# B&R Automation Studio project PLC code - cp (part 4)

#### ResetComms.st
```iecst
ACTION ResetComms:

	CanGetState.enable := TRUE;
	CanGetState.node := dataInv.Parameters.Hardware.Node;
	CanGetState.pDevice := ADR('SS1.IF1');
	CanGetState();

	iReasonNotComms.0 := CanGetState.state = coPREOPERATIONAL;
	iReasonNotComms.1 := CanGetState.state = coUNKNOWN;
	iReasonNotComms.2 := CanGetState.state = coNOTAVAIL;
	iReasonNotComms.3 := dataInv.Status.ErrorComms;

	tonNotComms.IN := iReasonNotComms > 0;
	tonNotComms.PT := t#3s;
	tonNotComms();

	xChangedResetCommsState := CanResetState_copy <> CanResetState;
	CanResetState_copy := CanResetState;

	CASE CanResetState OF

		COCOMSR_UNDEFINED,
		COCOMSR_COMMUNICATING:

			iTimesTryToReset := 0;

			//If time in error, define an error comms
			IF tonNotComms.Q THEN
				CanResetState := COCOMSR_COMMSERROR;
			END_IF

		COCOMSR_COMMSERROR:
			//Start the resetting process
			IF dataInv.Commands.Reset THEN //AND dataInv.Parameter.xAutoresetComms THEN
				//Communication has returned to work
				IF CanGetState.state = coOPERATIONAL THEN
					CanResetState := COCOMSR_COMMUNICATING;
				ELSE
					CanResetState := COCOMSR_RESETTING;
				END_IF
			END_IF

		COCOMSR_RESETTING:
			CANopenReset.enable := TRUE;
			CANopenReset.node := dataInv.Parameters.Hardware.Node;
			CANopenReset.pDevice := ADR('SS1.IF1');
			CANopenReset.state := coRESET_NODE;
			CANopenReset();

			IF CANopenReset.status = ERR_OK THEN
				lastCanOpenResetError := CANopenReset.error;
				CANopenReset(enable := FALSE);
				CanResetState := COCOMSR_WAITINGTOBERESETTED;
			END_IF

			tonCommsErrorResetting.IN := NOT xChangedResetCommsState;
			tonCommsErrorResetting.PT := t#10s;
			tonCommsErrorResetting();

			IF tonCommsErrorResetting.Q THEN
				lastResetingState := CanGetState.state;
				lastFbResetStatus := CANopenReset.status;
				tonCommsErrorResetting(IN:=FALSE);
				CANopenReset(enable:=FALSE);
				CanResetState := COCOMSR_RESETTING_ERROR;
			END_IF

		COCOMSR_WAITINGTOBERESETTED:

			//Communication has returned to work
			IF CanGetState.state = coOPERATIONAL THEN
				CanResetState := COCOMSR_COMMUNICATING;
			END_IF

			tonCommsErrorResetting.IN := NOT xChangedResetCommsState;
			tonCommsErrorResetting.PT := t#4s;
			tonCommsErrorResetting();

			IF tonCommsErrorResetting.Q THEN
				lastResetingState := CanGetState.state;
				lastFbResetStatus := CANopenReset.status;
				tonCommsErrorResetting(IN:=FALSE);
				CanResetState := COCOMSR_RESETTING_ERROR;
			END_IF

		COCOMSR_RESETTING_ERROR:

			//After an error, wait to try again
			tonCommsErrorResetting.IN := NOT xChangedResetCommsState;
			tonCommsErrorResetting.PT := t#500ms;
			tonCommsErrorResetting();

			IF tonCommsErrorResetting.Q  AND iTimesTryToReset < 6 THEN
				iTimesTryToReset := iTimesTryToReset + 1;
				CanResetState := COCOMSR_RESETTING;
			ELSIF tonCommsErrorResetting.Q THEN
				CanResetState := COCOMSR_COMMSERROR;
			END_IF

	END_CASE;

END_ACTION
```

#### Simulation.st
```iecst
ACTION Simulation:

	dataInv.Status.ErrorComms := FALSE;
	(********** Reset non appliant in simulation error flags **********)
	paramOk := TRUE;
	invalidHwAddress := FALSE;
	ioMap.In.ModuleOk := TRUE;
	connectionErrorNotAck := FALSE; //Uncomment for P66/P76
	(********** Inverter state machine **********)
	CASE StepSim OF
		STATE_NOT_READY_TO_SWITCH_ON:
			ioMap.In.StatusWord := 16#0000;
			IF ioMap.Out.ControlWord = 16#0000 THEN
				StepSim := STATE_SWITCH_ON_DISABLED;
			END_IF;

		STATE_SWITCH_ON_DISABLED:
			ioMap.In.StatusWord := 16#0040;
			IF ioMap.Out.ControlWord = 16#0006 THEN
				StepSim := STATE_READY_TO_SWITCH_ON;
			END_IF;

		STATE_READY_TO_SWITCH_ON:
			ioMap.In.StatusWord := 16#0021;
			IF ioMap.Out.ControlWord = 16#0007 THEN
				StepSim := STATE_SWITCHED_ON;
			ELSIF ioMap.Out.ControlWord = 16#0000 OR ioMap.Out.ControlWord = 16#0002 THEN
				StepSim := STATE_SWITCH_ON_DISABLED;
			END_IF;

		STATE_SWITCHED_ON:
			ioMap.In.StatusWord := 16#0023;
			IF ioMap.Out.ControlWord = 16#000F THEN
				StepSim := STATE_OPERATION_ENABLED;
			ELSIF ioMap.Out.ControlWord = 16#0006 THEN
				StepSim := STATE_READY_TO_SWITCH_ON;
			ELSIF ioMap.Out.ControlWord = 16#0000 OR ioMap.Out.ControlWord = 16#0002 THEN
				StepSim := STATE_SWITCH_ON_DISABLED;
			END_IF;

		STATE_OPERATION_ENABLED:
			ioMap.In.StatusWord := 16#0027;
			IF ioMap.Out.ControlWord = 16#0007 THEN
				StepSim := STATE_SWITCHED_ON;
			ELSIF ioMap.Out.ControlWord = 16#0006 THEN
				StepSim := STATE_READY_TO_SWITCH_ON;
			ELSIF ioMap.Out.ControlWord = 16#0000 OR ioMap.Out.ControlWord = 16#0002 THEN
				StepSim := STATE_SWITCH_ON_DISABLED;
			END_IF;

		STATE_QUICK_STOP_ACTIVE:
			ioMap.In.StatusWord := 16#0007;
			IF ioMap.Out.ControlWord = 16#0000 OR ioMap.Out.ControlWord = 16#0002 THEN
				StepSim := STATE_SWITCH_ON_DISABLED;
			END_IF;

		STATE_FAULT_REACTION_ACTIVE:
			ioMap.In.StatusWord := 16#000F;
			StepSim := STATE_FAULT;

		STATE_FAULT:
			ioMap.In.StatusWord := 16#0008;
			IF ioMap.Out.ControlWord = 16#0080 THEN
				StepSim := STATE_SWITCH_ON_DISABLED;
			END_IF;
	END_CASE;
	(********** Movement profile **********)
	IF StepSim = STATE_OPERATION_ENABLED THEN
		(* No decceleration parameter involved during operation *)
		SimDecceleration := 0;
		(* Acceleration and velocity calculation *)
		IF direction = 1 THEN
			IF REAL_TO_INT(SimVelocity) = UINT_TO_INT(dataInv.Parameters.Velocity) THEN
				SimAcceleration := 0;
			ELSIF REAL_TO_INT(SimVelocity) < UINT_TO_INT(dataInv.Parameters.Velocity) THEN
				SimAcceleration := UINT_TO_REAL(SimNominalSpeed) / dataInv.Parameters.AccelerationTime; (* positive acceleration in positive direction *)
				SimVelocity := LIMIT(-1*UINT_TO_REAL(SimNominalSpeed), SimInitialVelocity + SimVelocity + direction*(SimAcceleration * SimCycleTime), UINT_TO_REAL(dataInv.Parameters.Velocity));
			ELSIF REAL_TO_INT(SimVelocity) > UINT_TO_INT(dataInv.Parameters.Velocity) THEN
				SimAcceleration := -1*(UINT_TO_REAL(SimNominalSpeed) / dataInv.Parameters.AccelerationTime); (* negative acceleration in positive direction *)
				SimVelocity := LIMIT(UINT_TO_REAL(dataInv.Parameters.Velocity), SimInitialVelocity + SimVelocity + direction*(SimAcceleration * SimCycleTime), UINT_TO_REAL(SimNominalSpeed));
			END_IF;
		ELSIF direction = -1 THEN
			IF REAL_TO_INT(SimVelocity) = direction*UINT_TO_INT(dataInv.Parameters.Velocity) THEN
				SimAcceleration := 0;
			ELSIF REAL_TO_INT(SimVelocity) > direction*UINT_TO_INT(dataInv.Parameters.Velocity) THEN
				SimAcceleration := UINT_TO_REAL(SimNominalSpeed) / dataInv.Parameters.AccelerationTime; (* positive acceleration in negative direction *)
				SimVelocity := LIMIT(-1*UINT_TO_REAL(dataInv.Parameters.Velocity), SimInitialVelocity + SimVelocity + direction*(SimAcceleration * SimCycleTime), UINT_TO_REAL(SimNominalSpeed));
			ELSIF REAL_TO_INT(SimVelocity) < direction*UINT_TO_INT(dataInv.Parameters.Velocity) THEN
				SimAcceleration := -1*(UINT_TO_REAL(SimNominalSpeed) / dataInv.Parameters.AccelerationTime); (* negative acceleration in negative direction *)
				SimVelocity := LIMIT(-1*UINT_TO_REAL(SimNominalSpeed), SimInitialVelocity + SimVelocity + direction*(SimAcceleration * SimCycleTime), -1*UINT_TO_REAL(dataInv.Parameters.Velocity));
			END_IF;
		END_IF;
		(* Limiting the velocity to the nominal speed of the motor - Optional *)
		SimVelocity := LIMIT(-1*UINT_TO_REAL(SimNominalSpeed),SimVelocity,UINT_TO_REAL(SimNominalSpeed));

	ELSE
		(* No acceleration parameter involved during stop *)
		SimAcceleration := 0;
		(* Decceleration and velocity calculation *)
		IF REAL_TO_INT(SimVelocity) = 0 THEN
			SimDecceleration := 0;
		ELSIF REAL_TO_INT(SimVelocity) > 0 THEN
			SimDecceleration := -1*(UINT_TO_INT(SimNominalSpeed) / dataInv.Parameters.DecelerationTime);
			SimVelocity := LIMIT(0,SimInitialVelocity + SimVelocity + (SimDecceleration * SimCycleTime), UINT_TO_REAL(SimNominalSpeed));
		ELSIF REAL_TO_INT(SimVelocity) < 0 THEN
			SimDecceleration := UINT_TO_INT(SimNominalSpeed) / dataInv.Parameters.DecelerationTime;
			SimVelocity := LIMIT(-1*UINT_TO_REAL(SimNominalSpeed),SimInitialVelocity + SimVelocity + (SimDecceleration * SimCycleTime),0);
		END_IF;
	END_IF;
	ioMap.In.ActualSpeed :=  REAL_TO_INT(SimVelocity);
END_ACTION
```

### Package Logical/ExtPack/_Motion/StepperCtrl - Stepper Ctrl Logic package

### Package Logical/ExtPack/_Motion/StepperCtrl/StepperCtrl_v1 - Stepper Ctrl Logic package

### Program Logical/ExtPack/_Motion/StepperCtrl/StepperCtrl_v1/StepperX2XCtrl (IEC)

#### StepperX2XCtrl.st
```iecst
PROGRAM _CYCLIC

	//References
	pStepperCtrl ACCESS ADR(gAxisStepper[gIndexStepper]);

	IF NOT xInitDone THEN

		// initialize general interfaces
		IF gIndexStepper = 1 THEN
			// initialize general interfaces
			pStepperCtrl.gAxis.size  := pStepperCtrl.gAxis.size;
			pStepperCtrl.HW.DrvIf_Typ := ncSDC_DRVSM16;
			strcpy( ADR(pStepperCtrl.HW.DrvIf_Name[0]), ADR('gAxisStepper[1].DrvIf') );
			pStepperCtrl.HW.DiDoIf_Typ := ncSDC_DIDO;
			strcpy( ADR(pStepperCtrl.HW.DiDoIf_Name[0]), ADR('gAxisStepper[1].DiDoIf') );
			pStepperCtrl.HW.EncIf1_Typ := ncSDC_ENC16;
			strcpy( ADR(pStepperCtrl.HW.EncIf1_Name[0]), ADR('gAxisStepper[1].EncIf1') );
		END_IF;

		IF gIndexStepper = 2 THEN
			// initialize general interfaces
			pStepperCtrl.gAxis.size  := pStepperCtrl.gAxis.size;
			pStepperCtrl.HW.DrvIf_Typ := ncSDC_DRVSM16; //ncSDC_DRVSERVO16; -> To Servo control
			strcpy( ADR(pStepperCtrl.HW.DrvIf_Name[0]), ADR('gAxisStepper[2].DrvIf') );
			pStepperCtrl.HW.DiDoIf_Typ := ncSDC_DIDO;
			strcpy( ADR(pStepperCtrl.HW.DiDoIf_Name[0]), ADR('gAxisStepper[2].DiDoIf') );
			pStepperCtrl.HW.EncIf1_Typ := ncSDC_ENC16;
			strcpy( ADR(pStepperCtrl.HW.EncIf1_Name[0]), ADR('gAxisStepper[2].EncIf1') );
		END_IF;
		pStepperCtrl.EncIf1.iLifeCnt := pStepperCtrl.EncIf1.iLifeCnt;  //TOREVIEW. Can we remove it???

		// initialize old-value for delta step calculation

		oSetPosOld := pStepperCtrl.DrvIf.oSetPos;

		xInitDone := TRUE;
	END_IF

	(* life counter emulation of digital inputs *)
	pStepperCtrl.DiDoIf.iLifeCntReference := pStepperCtrl.DiDoIf.iLifeCntReference + 1;
	pStepperCtrl.DiDoIf.iLifeCntNegHwEnd  := pStepperCtrl.DiDoIf.iLifeCntNegHwEnd  + 1;
	pStepperCtrl.DiDoIf.iLifeCntPosHwEnd  := pStepperCtrl.DiDoIf.iLifeCntPosHwEnd  + 1;

	(* default function model of ACOPOSmicro: convert absolute steps to delta steps - overflow save delta calculation *)
	pStepperCtrl.MotorStep0 := pStepperCtrl.DrvIf.oSetPos - oSetPosOld;
	oSetPosOld := pStepperCtrl.DrvIf.oSetPos;

	gIndexStepper := gIndexStepper + 1;

END_PROGRAM
```

### Package Logical/ExtPack/_Motion/IclaCtrl - Icla Ctrl Logic package

### Package Logical/ExtPack/_Motion/IclaCtrl/IclaCtrl_v4 - Icla Ctrl Logic package

### Program Logical/ExtPack/_Motion/IclaCtrl/IclaCtrl_v4/IclaCtrl (IEC) - Icla Cyclic task

#### Variables.var
```iecst
VAR
	Icla : REFERENCE TO stIcla;
	PDO4 : REFERENCE TO IclaNetData_typ;
	StepIcla : stepAXISILE_enum := AXISILE_INIT;
	CANopenSDORead8_0 : CANopenSDORead8;
	CANopenSDORead8_1 : CANopenSDORead8; (*CANopenSDOWrite8_0 : CANopenSDOWrite8;*)
	CANopenSDORead8_2 : CANopenSDORead8;
	CANopenSDOWrite8_0 : CANopenSDOWrite8;
	CANopenSDOWrite8_2 : CANopenSDOWrite8;
	xOldInPosition : BOOL;
	xDebugIcla1 : BOOL := FALSE;
	xDebugIcla : BOOL := FALSE;
	iOutJogNoOrder : UINT;
	iOutJogOrderStop : UINT;
	uiCountJogOrders : UINT;
	xReadSpeed : BOOL;
	iPrevAcceleration : UINT;
	iPrevVeloSlow : UINT;
	iPrevVeloFast : UINT;
	StepComs : stepCOMSILE_enum;
	xEnabledReadComs : BOOL;
	xEnabledWriteComs : BOOL;
	xJogPauseSent : BOOL;
	uiValueToWrite : UINT; (*Value to write during debug in a register of datalen=2*)
	CanGetState : CANopenGetState;
	tonNotComms : TON;
	tonCommsErrorResetting : TON;
	CanResetState : CanOpenResetCommsState_enum;
	CanResetState_copy : CanOpenResetCommsState_enum;
	CANopenReset : CANopenNMT;
	iReasonNotComms : UINT;
	xChangedResetCommsState : BOOL;
	lastResetingState : UINT;
	lastFbResetStatus : UINT;
	lastCanOpenResetError : UINT;
	iTimesTryToReset : UINT;
END_VAR
VAR CONSTANT
	iHistoryLines : USINT := 20;
END_VAR
VAR
	StateHistory : ARRAY[0..iHistoryLines] OF stepAXISILE_enum;
	iIndexHistory : USINT;
END_VAR
```

#### Icla.st
```iecst
(*********************************************************************************
 * Copyright: Bernecker + Rainer
 * Author:		jorgemur
 * Created:		January 19, 2019
 * Version:		3.00.0
 * Description:	This task allows TO control an ICLA IFE motor through CANopen
				Manual movement, homing procedure, and MOVE absolute movements are
				implemented.
 *********************************************************************************)

PROGRAM _INIT
	StepIcla :=	AXISILE_INIT;
	StepComs := COMSILE_IDLE;
	xJogPauseSent:=FALSE;
	iPrevAcceleration:=2500;	//Defaul value in Icla. Just send the acceleration if it is changed by program
	iPrevVeloSlow:=300;			//Defaul value in Icla. Just send the acceleration if it is changed by program
	iPrevVeloFast:=1000;		//Defaul value in Icla. Just send the acceleration if it is changed by program
END_PROGRAM

PROGRAM _CYCLIC

	//IMPORTANT: When adding an ILE/ICLA motor on physical view. Copy and paste an existing one to get the device parameters required to get the motor enabled for operation
	Icla ACCESS ADR(gIcla[gIndexIcla]);
	PDO4 ACCESS ADR(gIclaNetData[gIndexIcla]);

	//Check drive status
	Icla.Status.iDriveStatus 		:= PDO4.TPDO4.driveStat AND 2#1111;
	Icla.Status.xReferenced 		:= PDO4.TPDO4.modeStat.5;
	Icla.Status.iActualPosition		:= PDO4.TPDO4.Act32;
	PDO4.RPDO4.driveCtrl.3 			:= Icla.Command.Reset;
	Icla.Status.xInPosition 		:= PDO4.TPDO4.driveStat.14;
	Icla.Status.xModuleOK			:= PDO4.xModuleOK;

	//Check communication status
	Icla.Status.Error.Communication := NOT Icla.Status.xModuleOK;

	//Limitation of the accepted values
	Icla.Parameter.Jog.VeloSlow 		 := LIMIT(300, Icla.Parameter.Jog.VeloSlow, 5000);
	Icla.Parameter.Jog.VeloFast 		 :=	LIMIT(300, Icla.Parameter.Jog.VeloFast, 5000);
	Icla.Parameter.MoveAbsolute.Velocity := LIMIT(300, Icla.Parameter.MoveAbsolute.Velocity, 5000);
	Icla.Parameter.iAcceleration 		 := LIMIT(1000, Icla.Parameter.iAcceleration, 10000);

	//	Start OF referencing mode action object: Write ACCESS triggers reference movement from
	//		1: LIMP
	//		2: LIMN
	//		3: REF neg. direction OF rotation
	//		4: REF pos. direction OF rotation
	//		7: Blocking movement neg. sense OF rotation
	//		8: Blocking movement pos. sense OF rotation
	//	Icla.Parameter.Home.Mode = LIMIT(0,Icla.Parameter.Home.Mode,8)
	//	IF Icla.Parameter.Home.Mode = 5 OR Icla.Parameter.Home.Mode = 6 THEN
	//		Icla.Parameter.Home.Mode = :=0;
	//	END_IF

	CASE StepIcla OF

		AXISILE_INIT:

			IF iPrevAcceleration = Icla.Parameter.iAcceleration AND
				iPrevVeloSlow = Icla.Parameter.Jog.VeloSlow AND
				(iPrevVeloFast = Icla.Parameter.Jog.VeloFast OR NOT Icla.Command.JogFastSpeed)AND
				xJogPauseSent 										THEN
				StepIcla := AXISILE_WAIT_READY_TO_SWITCH_ON;
			END_IF

		AXISILE_WAIT_READY_TO_SWITCH_ON:
			Icla.Status.Info := 'Waiting for enable input';
			//Reset commands
			Icla.Command.Home := FALSE;
			Icla.Command.MoveAbsolute := FALSE;
			Icla.Command.JogBackward := FALSE;
			Icla.Command.JogForward := FALSE;
			Icla.Command.JogFastSpeed := FALSE;
			Icla.Command.Stop := FALSE;
			Icla.Command.Reset := FALSE;

			//Reset mode
			PDO4.RPDO4.modeCtrl := 0;

			PDO4.RPDO4.driveCtrl.0 := TRUE;//Disable Power
			PDO4.RPDO4.driveCtrl.1 := FALSE;//Enable Power

			IF Icla.Status.iDriveStatus = 3  THEN
				PDO4.RPDO4.driveCtrl.0 := TRUE;//Disable Power
				PDO4.RPDO4.driveCtrl.1 := FALSE;//Enable Power
				//TOJMH: Review 4 & 6 or just 4 (And 6 for AXISILE_READY)
			ELSIF Icla.Status.iDriveStatus = 4 OR Icla.Status.iDriveStatus = 6 THEN
				StepIcla := AXISILE_WAIT;
				//TOJMH: Review when QuickStop appears
			ELSIF Icla.Status.iDriveStatus = 7 THEN	//Go out of state 7 (quick stop)
				Icla.Command.Reset := TRUE;
			END_IF

			//Toggle to send data
			PDO4.RPDO4.modeCtrl.7	:= NOT PDO4.TPDO4.modeStat.7;

		AXISILE_WAIT:
			Icla.Status.Info := 'Waiting for enable command';
			//Reset commands
			Icla.Command.Home := FALSE;
			Icla.Command.MoveAbsolute := FALSE;
			Icla.Command.JogBackward := FALSE;
			Icla.Command.JogForward := FALSE;
			Icla.Command.JogFastSpeed := FALSE;
			Icla.Command.Stop := FALSE;

			//Reset mode
			PDO4.RPDO4.modeCtrl := 0;

			IF Icla.Command.Enable THEN
				PDO4.RPDO4.driveCtrl.0 := FALSE;//Disable Power
				PDO4.RPDO4.driveCtrl.1 := TRUE;//Enable Power
			ELSE
				PDO4.RPDO4.driveCtrl.0 := TRUE;//Disable Power
				PDO4.RPDO4.driveCtrl.1 := FALSE;//Enable Power
			END_IF;
			IF Icla.Command.Enable AND Icla.Status.iDriveStatus = ICLAST_ENABLE_OPERATION  THEN
				StepIcla := AXISILE_POWER;
			ELSIF Icla.Status.iDriveStatus = 3  THEN
				StepIcla := AXISILE_WAIT_READY_TO_SWITCH_ON;
			ELSIF Icla.Status.iDriveStatus = 7 THEN	//Go out of state 7 (quick stop)
				Icla.Command.Reset := TRUE;
				Icla.Command.Enable := FALSE; //Due to issue DELOREAN-746
			END_IF;

			//Toggle to send data
			PDO4.RPDO4.modeCtrl.7	:= NOT PDO4.TPDO4.modeStat.7;

		AXISILE_POWER:
			Icla.Status.Info := 'Waiting for power on';
			//Reset commands

			//Reset commands
			Icla.Command.MoveAbsolute := FALSE;
			Icla.Command.Reset := FALSE;
			Icla.Command.Stop := FALSE;

			IF NOT Icla.Command.Enable THEN
				PDO4.RPDO4.driveCtrl.0 := TRUE;//Disable Power
				PDO4.RPDO4.driveCtrl.1 := FALSE;//Enable Power
				StepIcla :=AXISILE_WAIT_READY_TO_SWITCH_ON;
			END_IF;

			IF Icla.Status.xReferenced THEN
				StepIcla := AXISILE_READY;
			END_IF

			IF Icla.Command.Home  THEN
				IF NOT Icla.Status.xReferenced THEN
					StepIcla := AXISILE_HOMING;
				END_IF;
			ELSIF Icla.Command.JogBackward OR Icla.Command.JogForward THEN
				StepIcla := AXISILE_JOG;
			END_IF;

			//Toggle to send data
			PDO4.RPDO4.modeCtrl.7	:= NOT PDO4.TPDO4.modeStat.7;

		AXISILE_HOMING:

			//Reset commands
			//Icla.Command.Enable := TRUE;
			Icla.Command.Home := FALSE;
			Icla.Command.MoveAbsolute := FALSE;
			Icla.Command.JogBackward := FALSE;
			Icla.Command.JogForward := FALSE;
			Icla.Command.JogFastSpeed := FALSE;
			Icla.Command.Reset := FALSE;
			Icla.Command.Stop := FALSE;

			//Mode = 2, HOMING
			PDO4.RPDO4.modeCtrl.2	:= FALSE;
			PDO4.RPDO4.modeCtrl.1	:= TRUE;
			PDO4.RPDO4.modeCtrl.0	:= FALSE;

			//Action = 0, DIMENSION SETTING
			IF Icla.Parameter.Home.Mode = 0 THEN	//Dimension setting
				PDO4.RPDO4.modeCtrl.6	:= FALSE;
				PDO4.RPDO4.modeCtrl.5	:= FALSE;
				PDO4.RPDO4.modeCtrl.4	:= FALSE;
				PDO4.RPDO4.Ref32 		:= Icla.Parameter.Home.Position;
			ELSE
				PDO4.RPDO4.modeCtrl.6	:= FALSE;
				PDO4.RPDO4.modeCtrl.5	:= FALSE;
				PDO4.RPDO4.modeCtrl.4	:= TRUE;
				PDO4.RPDO4.Ref16 		:= Icla.Parameter.Home.Mode;
			END_IF;
			(* Start of referencing mode action object: Write ACCESS triggers reference movement from
				1: LIMP
				2: LIMN
				3: REF neg. direction OF rotation
				4: REF pos. direction OF rotation
				7: Blocking movement neg. sense OF rotation
				8: Blocking movement pos. sense OF rotation
			*)

			//Check if Referenced is done. Prior to send data
			IF Icla.Status.xReferenced AND EDGE(PDO4.TPDO4.modeStat.7) THEN
				StepIcla := AXISILE_READY;
			END_IF;

			//Toggle to send data
			PDO4.RPDO4.modeCtrl.7	:= NOT PDO4.TPDO4.modeStat.7;

		AXISILE_READY:
			//Reset commands
			Icla.Command.Stop := FALSE;
			Icla.Status.Info := 'Ready to perform movements';
			IF Icla.Command.JogBackward OR Icla.Command.JogForward THEN
				Icla.Status.xInPosition := FALSE;
				StepIcla := AXISILE_JOG;
				uiCountJogOrders:=uiCountJogOrders+1;
			ELSIF Icla.Command.MoveAbsolute THEN
				IF Icla.Status.iActualPosition <> Icla.Parameter.MoveAbsolute.Position THEN
					StepIcla := AXISILE_MOVE_ABSOLUTE;
				ELSE
					Icla.Command.MoveAbsolute := FALSE;
				END_IF;

			ELSIF NOT Icla.Command.Enable THEN
				Icla.Status.xInPosition := FALSE;
				StepIcla := AXISILE_WAIT_READY_TO_SWITCH_ON;
			ELSIF Icla.Command.Home THEN
				Icla.Status.xInPosition := FALSE;
				StepIcla := AXISILE_HOMING;
			END_IF;

		AXISILE_JOG:
			Icla.Status.Info := 'Jogging';
			//Reset commands
			//Icla.Command.Enable := TRUE;
			Icla.Command.MoveAbsolute := FALSE;
			Icla.Command.Home := FALSE;
			Icla.Command.Reset := FALSE;

			PDO4.RPDO4.modeCtrl := 1;	//Manual mode

			IF Icla.Command.JogBackward AND Icla.Command.JogForward THEN
				Icla.Command.JogBackward := FALSE;
				Icla.Command.JogForward  := FALSE;
			END_IF;
			//Jog negative
			IF Icla.Command.JogBackward THEN
				Icla.Command.JogForward := FALSE;
				PDO4.RPDO4.Ref16.0 := FALSE;
				PDO4.RPDO4.Ref16.1 := TRUE;
				PDO4.RPDO4.Ref16.2 := Icla.Command.JogFastSpeed;
			END_IF
			//Jog positive
			IF Icla.Command.JogForward THEN
				Icla.Command.JogBackward := FALSE;
				PDO4.RPDO4.Ref16.0 := TRUE;
				PDO4.RPDO4.Ref16.1 := FALSE;
				PDO4.RPDO4.Ref16.2 := Icla.Command.JogFastSpeed;
			END_IF;
			IF NOT Icla.Command.JogBackward AND NOT Icla.Command.JogForward THEN
				PDO4.RPDO4.Ref16.0 := FALSE;
				PDO4.RPDO4.Ref16.1 := FALSE;
				PDO4.RPDO4.Ref16.2 := FALSE;
				IF Icla.Status.iActualVelocity=0 THEN
					StepIcla := AXISILE_WAIT_READY_TO_SWITCH_ON;
				END_IF
				iOutJogNoOrder:=iOutJogNoOrder+1;
			END_IF;
			//Send Quick-Stop command
			IF Icla.Command.Stop THEN
				Icla.Command.JogBackward	:= FALSE;
				Icla.Command.JogForward	:= FALSE;
				PDO4.RPDO4.Ref16.0			:= FALSE;
				PDO4.RPDO4.Ref16.1			:= FALSE;
				PDO4.RPDO4.Ref16.2			:= FALSE;
				PDO4.RPDO4.driveCtrl.2		:= TRUE;//QuickStop
				StepIcla := AXISILE_WAIT_READY_TO_SWITCH_ON;
				iOutJogOrderStop:=iOutJogOrderStop+1;
			END_IF
			//Toggle to send data
			PDO4.RPDO4.modeCtrl.7	:= NOT 	PDO4.TPDO4.modeStat.7;

		AXISILE_MOVE_ABSOLUTE:
			IF Icla.Parameter.MoveAbsolute.Velocity = 0 THEN
				Icla.Status.Info := 'WARNING: set speed is 0, please change it';
			ELSE
				Icla.Status.Info := 'Moving to set position';
			END_IF;

			//Reset commands
			//Icla.Command.Enable := TRUE;
			Icla.Command.Home := FALSE;
			Icla.Command.JogBackward := FALSE;
			Icla.Command.JogForward := FALSE;
			Icla.Command.JogFastSpeed := FALSE;
			Icla.Command.MoveAbsolute := TRUE;

			//Setpoint Speed
			PDO4.RPDO4.Ref16 := Icla.Parameter.MoveAbsolute.Velocity;
			//Setpoint Position
			PDO4.RPDO4.Ref32 := Icla.Parameter.MoveAbsolute.Position;

			//Mode = 3, PTP
			PDO4.RPDO4.modeCtrl.2	:= FALSE;
			PDO4.RPDO4.modeCtrl.1	:= TRUE;
			PDO4.RPDO4.modeCtrl.0	:= TRUE;

			//Action = 0, ABSOLUTE POSITIONING
			PDO4.RPDO4.modeCtrl.6	:= FALSE;
			PDO4.RPDO4.modeCtrl.5	:= FALSE;
			PDO4.RPDO4.modeCtrl.4	:= FALSE;

			//Toggle to send data
			PDO4.RPDO4.modeCtrl.7	:= NOT 	PDO4.TPDO4.modeStat.7;

			//Rising edge in InPosition to jump to READY
			IF Icla.Status.xInPosition AND NOT xOldInPosition THEN
				StepIcla := AXISILE_WAIT;
			END_IF

			IF NOT Icla.Command.Enable THEN
				Icla.Status.xInPosition := FALSE;
				StepIcla := AXISILE_WAIT_READY_TO_SWITCH_ON;
			END_IF

			IF Icla.Command.Stop THEN		//Send Quick-Stop command
				Icla.Command.JogBackward	:= FALSE;
				Icla.Command.JogForward	:= FALSE;
				PDO4.RPDO4.Ref16.0			:= FALSE;
				PDO4.RPDO4.Ref16.1			:= FALSE;
				PDO4.RPDO4.Ref16.2			:= FALSE;
				PDO4.RPDO4.driveCtrl.2		:= TRUE;//QuickStop
				StepIcla := AXISILE_WAIT_READY_TO_SWITCH_ON;
			END_IF

		AXISILE_ERROR:

			IF Icla.Status.Info <> 'ERROR transfering Jog parameters' THEN
				Icla.Status.Info := 'ERROR';
			END_IF;
			//Reset commands
			Icla.Command.Enable := FALSE;
			Icla.Command.Home := FALSE;
			Icla.Command.MoveAbsolute := FALSE;
			Icla.Command.JogBackward := FALSE;
			Icla.Command.JogForward := FALSE;
			Icla.Command.JogFastSpeed := FALSE;
			Icla.Command.Stop := FALSE;

			//Reseting errors
			PDO4.RPDO4.driveCtrl.3 := Icla.Command.Reset;

			IF Icla.Command.Reset (*AND Icla.Status.iDriveStatus <> ICLAST_ERROR*) THEN
				Icla.Status.Error.Jog := FALSE;
				Icla.Status.Error.ErrorNumber := 0;
				StepIcla := AXISILE_WAIT_READY_TO_SWITCH_ON;
			END_IF

	END_CASE

	ResetComms;

	xReadSpeed := Icla.Status.iActualVelocity<>0; // AND NOT Icla.Status.xInError;

	IclaSDO;

	//ERROR handling
	IF StepIcla <> AXISILE_INIT AND (EDGEPOS(Icla.Status.iDriveStatus = ICLAST_ERROR) OR Icla.Status.Error.Communication OR Icla.Status.Error.Jog) THEN
		StepIcla := AXISILE_ERROR;
	END_IF

	Icla.Status.xInError := StepIcla = AXISILE_ERROR;

	//Icla state story
	IF StepIcla<>StateHistory[0] THEN
		FOR iIndexHistory:=iHistoryLines TO 1 BY -1 DO
			StateHistory[iIndexHistory]:=StateHistory[iIndexHistory-1];
		END_FOR
		StateHistory[0]:=StepIcla;
	END_IF

	xOldInPosition := Icla.Status.xInPosition;

	Icla.Status.IclaStatus:=StepIcla;
	Icla.Status.IclaSDOStep:=StepComs;

	// After all tasks, incr and sanity check
	gIndexIcla := gIndexIcla + 1;

END_PROGRAM
```

#### IclaSDO.st
```iecst
ACTION IclaSDO:

	// COMMS COMMS COMMS COMMS COMMS COMMS COMMS COMMS COMMS COMMS COMMS COMMS COMMS COMMS COMMS COMMS COMMS COMMS COMMS COMMS
	// COMMS COMMS COMMS COMMS COMMS COMMS COMMS COMMS COMMS COMMS COMMS COMMS COMMS COMMS COMMS COMMS COMMS COMMS COMMS COMMS
	// COMMS COMMS COMMS COMMS COMMS COMMS COMMS COMMS COMMS COMMS COMMS COMMS COMMS COMMS COMMS COMMS COMMS COMMS COMMS COMMS

	// IMPORTANT NOTE!!  && && && && && && && && && && && && && && && && && &&
	//
	// The Index to be sent in the SDO functions is in the form 16#30xx, where xx is the index in the manual in HEX code
	//
	// IMPORTANT NOTE!!  && && && && && && && && && && && && && && && && && &&

	CANopenSDOWrite8_0.enable := xEnabledWriteComs;
	CANopenSDOWrite8_0.pDevice := ADR(Icla.Parameter.Network);
	CANopenSDOWrite8_0.node := Icla.Parameter.Node;

	CANopenSDORead8_1.pDevice := ADR(Icla.Parameter.Network);
	CANopenSDORead8_1.node := Icla.Parameter.Node;

	CASE StepComs OF
		COMSILE_IDLE:
			IF Icla.Parameter.Node = 255 THEN
				//Waiting to be configured or errors removed
			ELSIF StepIcla = AXISILE_JOG OR StepIcla = AXISILE_MOVE_ABSOLUTE OR xReadSpeed THEN
				StepComs := COMSILE_READ_SPEED;
//			ELSIF StepIcla=AXISILE_ERROR THEN
//				StepComs := COMSILE_ERROR;
			ELSIF StepIcla <> AXISILE_ERROR AND StepComs = COMSILE_ERROR THEN
				StepComs := COMSILE_IDLE;
			ELSIF NOT xJogPauseSent THEN
				StepComs := COMSILE_JOG_PAUSE;
			ELSIF iPrevAcceleration <> Icla.Parameter.iAcceleration THEN
				StepComs := COMSILE_ACCELERATION;
			ELSIF iPrevVeloSlow <> Icla.Parameter.Jog.VeloSlow THEN
				StepComs := COMSILE_JOG_TRANSFER_SLOW;
			ELSIF (iPrevVeloFast <> Icla.Parameter.Jog.VeloFast) AND Icla.Command.JogFastSpeed THEN
				StepComs := COMSILE_JOG_TRANSFER_FAST;
			END_IF

		COMSILE_JOG_PAUSE:
			CANopenSDOWrite8_0.data0 := 0;
			CANopenSDOWrite8_0.data1 := 0;
			CANopenSDOWrite8_0.datalen := 2;
			CANopenSDOWrite8_0.index := 16#3029;
			CANopenSDOWrite8_0.subindex := 16#07;
			CANopenSDOWrite8_0.enable:=TRUE;
			CANopenSDOWrite8_0();

			IF CANopenSDOWrite8_0.status = ERR_OK THEN
				Icla.Command.Reset := TRUE;  //To avoid starting with the Icla in error state
				StepComs := COMSILE_IDLE;
				xJogPauseSent:=TRUE;
				CANopenSDOWrite8_0.enable:=FALSE;
			ELSIF CANopenSDOWrite8_0.status <> ERR_FUB_BUSY AND CANopenSDOWrite8_0.status <> ERR_FUB_ENABLE_FALSE THEN
				Icla.Status.Info := 'ERROR transfering Jog Pause parameter';
				CANopenSDOWrite8_0.enable:=FALSE;
			END_IF;

		COMSILE_ACCELERATION:
			CANopenSDOWrite8_0.data0 := UINT_TO_USINT(Icla.Parameter.iAcceleration AND 16#00FF);
			CANopenSDOWrite8_0.data1 := UINT_TO_USINT(SHR((Icla.Parameter.iAcceleration AND 16#FF00),8));
			CANopenSDOWrite8_0.data2 := 0;
			CANopenSDOWrite8_0.data3 := 0;
			CANopenSDOWrite8_0.datalen := 4;
			CANopenSDOWrite8_0.index := 16#301D;
			CANopenSDOWrite8_0.subindex := 16#1A;
			CANopenSDOWrite8_0.enable:=TRUE;
			CANopenSDOWrite8_0();

			IF CANopenSDOWrite8_0.status = ERR_OK THEN
				StepComs := COMSILE_IDLE;
				iPrevAcceleration := Icla.Parameter.iAcceleration;
				CANopenSDOWrite8_0.enable:=FALSE;
			ELSIF CANopenSDOWrite8_0.status <> ERR_FUB_BUSY AND CANopenSDOWrite8_0.status <> ERR_FUB_ENABLE_FALSE THEN
				Icla.Status.Info := 'ERROR transfering Acceleration parameter';
				CANopenSDOWrite8_0.enable:=FALSE;
			END_IF;

		COMSILE_JOG_TRANSFER_SLOW:
			CANopenSDOWrite8_0.data0 := UINT_TO_USINT(Icla.Parameter.Jog.VeloSlow AND 16#00FF);
			CANopenSDOWrite8_0.data1 := UINT_TO_USINT(SHR((Icla.Parameter.Jog.VeloSlow AND 16#FF00),8));
			CANopenSDOWrite8_0.datalen := 2;
			CANopenSDOWrite8_0.index := 16#3029;
			CANopenSDOWrite8_0.subindex := 16#04;
			CANopenSDOWrite8_0.enable:=TRUE;
			CANopenSDOWrite8_0();

			IF CANopenSDOWrite8_0.status = ERR_OK THEN
				StepComs := COMSILE_IDLE;
				iPrevVeloSlow := Icla.Parameter.Jog.VeloSlow;
				CANopenSDOWrite8_0.enable:=FALSE;
			ELSIF CANopenSDOWrite8_0.status <> ERR_FUB_BUSY AND CANopenSDOWrite8_0.status <> ERR_FUB_ENABLE_FALSE THEN
				Icla.Status.Info := 'ERROR transfering Jog Slow Speed parameter';
				CANopenSDOWrite8_0.enable:=FALSE;
			END_IF;

		COMSILE_JOG_TRANSFER_FAST:
			CANopenSDOWrite8_0.data0 := UINT_TO_USINT(Icla.Parameter.Jog.VeloFast AND 16#00FF);
			CANopenSDOWrite8_0.data1 := UINT_TO_USINT(SHR((Icla.Parameter.Jog.VeloFast AND 16#FF00),8));
			CANopenSDOWrite8_0.datalen := 2;
			CANopenSDOWrite8_0.index := 16#3029;
			CANopenSDOWrite8_0.subindex := 16#05;
			CANopenSDOWrite8_0.enable:=TRUE;
			CANopenSDOWrite8_0();

			IF CANopenSDOWrite8_0.status = ERR_OK THEN
				StepComs := COMSILE_IDLE;
				iPrevVeloFast := Icla.Parameter.Jog.VeloFast;
				CANopenSDOWrite8_0.enable:=FALSE;
			ELSIF CANopenSDOWrite8_0.status <> ERR_FUB_BUSY AND CANopenSDOWrite8_0.status <> ERR_FUB_ENABLE_FALSE THEN
				Icla.Status.Info := 'ERROR transfering Jog Fast Speed parameter';
				CANopenSDOWrite8_0.enable:=FALSE;
			END_IF;

		COMSILE_READ_SPEED:
			//Read motor speed
			CANopenSDORead8_1.index := 16#301F;
			CANopenSDORead8_1.subindex := 16#09;
			CANopenSDORead8_1.enable := NOT Icla.Command.Reset;
			CANopenSDORead8_1();
			Icla.Status.iActualVelocity := SHL(USINT_TO_UINT(CANopenSDORead8_1.data1),8) + USINT_TO_UINT(CANopenSDORead8_1.data0);
			IF StepIcla <> AXISILE_JOG AND StepIcla <> AXISILE_MOVE_ABSOLUTE THEN
				StepComs := COMSILE_IDLE;
				CANopenSDORead8_1.enable:=FALSE;
				CANopenSDORead8_1();
				//Icla.Status.iActualVelocity := 0;
			END_IF

		COMSILE_ERROR:
			//Read error number
			CANopenSDORead8_0.index := 16#3020;
			CANopenSDORead8_0.subindex := 16#07;
			CANopenSDORead8_0.enable := NOT Icla.Command.Reset;
			CANopenSDORead8_0();
			IF CANopenSDORead8_0.status = ERR_OK THEN
				Icla.Status.Error.ErrorNumber := SHL(USINT_TO_UINT(CANopenSDORead8_0.data1),8) + USINT_TO_UINT(CANopenSDORead8_0.data0);
				IF Icla.Status.Error.ErrorNumber=0 AND StepIcla <> AXISILE_ERROR THEN
					StepComs:=COMSILE_IDLE;
				END_IF
				//After communicating, leave the channel free to the next communication
				CANopenSDORead8_0.enable := FALSE;
				CANopenSDORead8_0();
			ELSIF CANopenSDORead8_0.status <> ERR_FUB_BUSY THEN
				StepComs:=COMSILE_IDLE;
				//After communicating, leave the channel free to the next communication
				CANopenSDORead8_0.enable := FALSE;
				CANopenSDORead8_0();
			END_IF;

			IF Icla.Command.Reset AND Icla.Status.iDriveStatus <> ICLAST_ERROR THEN
				CANopenSDORead8_0.enable := FALSE;
				CANopenSDORead8_0();
			END_IF;

	END_CASE;

	///////////////////////////////////////////////////////////////////////////////

	//Limitation of Icla.Parameter.writeRegister.TotalBytes. Just 2 and 4 are valid values
	Icla.Parameter.writeRegister.TotalBytes:= LIMIT(2, Icla.Parameter.writeRegister.TotalBytes, 4);
	IF Icla.Parameter.writeRegister.TotalBytes = 3 THEN Icla.Parameter.writeRegister.TotalBytes:=2; END_IF

	//If Comms are not in idle is because we are communicating
	IF StepComs <> COMSILE_IDLE THEN

		Icla.Status.readRegister.xDataOK:=FALSE;

		CANopenSDOWrite8_2.enable := FALSE;
		CANopenSDOWrite8_2();
		CANopenSDORead8_0.enable := FALSE;
		CANopenSDORead8_0();
		CANopenSDORead8_2.enable := FALSE;
		CANopenSDORead8_2();

		RETURN;
	END_IF

	CANopenSDOWrite8_2.enable := Icla.Parameter.writeRegister.WriteOrder AND NOT CANopenSDORead8_2.enable;
	CANopenSDOWrite8_2.pDevice := ADR(Icla.Parameter.Network);
	CANopenSDOWrite8_2.node := Icla.Parameter.Node;
	IF CANopenSDOWrite8_2.enable THEN
		//CANopenSDOWrite8_2.data0 := UINT_TO_USINT(uiValueToWrite AND 16#00FF);
		//CANopenSDOWrite8_2.data1 := UINT_TO_USINT(SHR((uiValueToWrite AND 16#FF00),8));
		CANopenSDOWrite8_2.data0 := Icla.Parameter.writeRegister.data.data0;
		CANopenSDOWrite8_2.data1 := Icla.Parameter.writeRegister.data.data1;
		CANopenSDOWrite8_2.data2 := Icla.Parameter.writeRegister.data.data2;
		CANopenSDOWrite8_2.data3 := Icla.Parameter.writeRegister.data.data3;
		CANopenSDOWrite8_2.datalen := Icla.Parameter.writeRegister.TotalBytes;
		CANopenSDOWrite8_2.index := 16#3000 OR USINT_TO_UINT(Icla.Parameter.writeRegister.writeRegister.index);
		CANopenSDOWrite8_2.subindex := Icla.Parameter.writeRegister.writeRegister.subindex;
		Icla.Status.writeRegisterOK:=FALSE;
	END_IF
	CANopenSDOWrite8_2();

	IF CANopenSDOWrite8_2.status = ERR_OK THEN
		Icla.Parameter.writeRegister.WriteOrder:=FALSE;
		Icla.Status.writeRegisterOK:=TRUE;
	ELSIF CANopenSDOWrite8_2.status <> ERR_FUB_BUSY AND CANopenSDOWrite8_2.status <> ERR_FUB_ENABLE_FALSE THEN
		Icla.Status.Info := 'ERROR Writing Registers';
		Icla.Parameter.writeRegister.WriteOrder:=FALSE;
	END_IF;

	CANopenSDORead8_2.enable := NOT CANopenSDORead8_0.enable AND NOT CANopenSDORead8_1.enable AND NOT CANopenSDOWrite8_0.enable AND NOT Icla.Parameter.writeRegister.WriteOrder;
	CANopenSDORead8_2.pDevice := ADR(Icla.Parameter.Network);
	CANopenSDORead8_2.node := Icla.Parameter.Node;
	CANopenSDORead8_2.index := 16#3000 OR USINT_TO_UINT(Icla.Parameter.readRegister.index);
	CANopenSDORead8_2.subindex := Icla.Parameter.readRegister.subindex;
	CANopenSDORead8_2();
	Icla.Status.readRegister.xBusy := CANopenSDORead8_2.status <> ERR_FUB_BUSY;
	IF CANopenSDORead8_2.status = ERR_OK THEN
		Icla.Status.readRegister.xDataOK:=TRUE;
		Icla.Status.readRegister.rawData.data0:=CANopenSDORead8_2.data0;
		Icla.Status.readRegister.rawData.data1:=CANopenSDORead8_2.data1;
		Icla.Status.readRegister.rawData.data2:=CANopenSDORead8_2.data2;
		Icla.Status.readRegister.rawData.data3:=CANopenSDORead8_2.data3;
		Icla.Status.readRegister.uiValue := SHL(USINT_TO_UINT(CANopenSDORead8_2.data1),8) + USINT_TO_UINT(CANopenSDORead8_2.data0);
		Icla.Status.readRegister.usiValue := CANopenSDORead8_2.data0;
	ELSIF CANopenSDORead8_2.status <> ERR_FUB_BUSY AND CANopenSDORead8_2.status <> ERR_FUB_ENABLE_FALSE THEN
		Icla.Status.Info := 'ERROR Reading Registers';
		Icla.Status.readRegister.xDataOK:=FALSE;
		Icla.Status.readRegister.rawData.data0:=0;
		Icla.Status.readRegister.rawData.data1:=0;
		Icla.Status.readRegister.rawData.data2:=0;
		Icla.Status.readRegister.rawData.data3:=0;
		Icla.Status.readRegister.uiValue := 0;
		Icla.Status.readRegister.usiValue := 0;
	END_IF;

END_ACTION
```

#### ReadmeIcla.txt
```
	(* From Icla datasheet

	Motor.Status.DriveStatu = 4 -> Ready TO Switch On off Passive operating state,
	motor without current
	Motor.Status.DriveStatu = 6  -> Operation Enable on Active operating state, current
	available TO motor
	Motor.Status.DriveStatu = 7 -> Quick Stop active on Fault state, power stage
	remains enabled
	Motor.Status.DriveStatu = 9 -> Fault off Fault state, power stage is
	disabled

	The field drivectrl in the object: PDO4.RPDO4.driveCtrl
	Bit no. Value Meaning
	0 01h Disable
	1 02h Enable
	2 04h Quick Stop
	3 08h Fault Reset
	4 10h Quick Stop release

	R_PDO4 provides three fields FOR these purposes:
	• modeCtrl Starting AND changing operating modes
	• "Ref16" AND "Ref32" Operating mode-dependent reference values
	The specified values FOR these three fields are NOT taken over BY the product
	UNTIL modeCtrl, bit 7 (ModeToggle) changes

	IF the product was originally in operating state 9, it will switch TO operating
	state 4 after the "Fault Reset". You THEN have TO transmit a "0 -> 1" EDGE
	in drivectrl, bit 1 "Enable", in order TO enable the power stage.

	drivectrl:
	Bit 0: Power stage Disable Triggered when 0 changes TO 1 Triggered at write ACCESS IF bit value = 1
	Bit 1: Power stage Enable
	Bit 2: Quickstop
	Bit 3: Fault Reset
	Bit 4: Quickstop Release
	*)
```

### Program Logical/ExtPack/_Motion/IclaCtrl/IclaCtrl_v4/InitIclaCtrl (IEC) - Handling Index Icla

#### InitIclaIndex.st - Index code
```iecst
PROGRAM _CYCLIC
	gIndexIcla	:= 1;

END_PROGRAM
```

### Icla.var - Global Icla vars
```iecst
VAR
	gIndexIcla : USINT;
END_VAR
```

- IclaStates.graphml - IclaStates (not shown)

### IclaSim.typ
```iecst
TYPE
	stIclaParameters : 	STRUCT
		SpeedFactor : REAL := 1.0; (*The modification of the speed configured to speed up simulations*)
	END_STRUCT;
	stIclaSim : 	STRUCT
		Parameters : stIclaParameters;
	END_STRUCT;
END_TYPE
```

### IclaSimGen.var
```iecst
VAR
	iIclaSimIndex : USINT;
END_VAR
```

### Program Logical/ExtPack/_Motion/IclaCtrl/IclaSim/IclaSim_v1/IclaSim (IEC)

#### Main.st - Init, cyclic, exit code
```iecst
//ncAbsMov := ncHALT_OK;

PROGRAM _CYCLIC

	Icla ACCESS ADR(gIcla[iIclaSimIndex]);
	IclaSim ACCESS ADR(gIclaSim[iIclaSimIndex]);

	IF NOT Icla.Command.Enable THEN
		ncAbsMov := ncHALT_OK;
		Icla.Status.iActualVelocity := 0;
		Icla.Status.IclaStatus:= AXISILE_WAIT;
		iIclaSimIndex := iIclaSimIndex + 1;
		RETURN;
	END_IF

	//Home the Icla
	IF EDGEPOS(Icla.Command.Home) THEN
		Icla.Status.xReferenced:=TRUE;
		Icla.Status.iActualPosition:=Icla.Parameter.Home.Position;
		rActPosition := DINT_TO_REAL(Icla.Status.iActualPosition);
		Icla.Command.Home:=FALSE;
	END_IF

	IF Icla.Command.JogBackward AND Icla.Command.JogForward THEN
		Icla.Command.JogBackward:=FALSE;
		Icla.Command.JogForward:=FALSE;
	END_IF

	//Defining the advance in each direction and the stop
	rMsFromLastExec := TIME_TO_REAL(clock_ms()-tiLastExec);

	IF Icla.Command.JogBackward THEN
		IF Icla.Command.JogFastSpeed THEN
			//Define the advance. The minimum advance will be 1. The speed is defined in revs per minute
			rAdvance := IclaSim.Parameters.SpeedFactor * UINT_TO_REAL(Icla.Parameter.Jog.VeloFast)*rMsFromLastExec/1000;
		ELSE
			//Define the advance. The minimum advance will be 1. The speed is defined in revs per minute
			rAdvance := IclaSim.Parameters.SpeedFactor * UINT_TO_REAL(Icla.Parameter.Jog.VeloSlow)*rMsFromLastExec/1000;
		END_IF
		rActPosition := rActPosition - rAdvance;
		Icla.Status.iActualPosition := REAL_TO_DINT(rActPosition);
	END_IF

	IF Icla.Command.JogForward THEN
		IF Icla.Command.JogFastSpeed THEN
			//Define the advance. The minimum advance will be 1. The speed is defined in revs per minute
			rAdvance := IclaSim.Parameters.SpeedFactor * UINT_TO_REAL(Icla.Parameter.Jog.VeloFast)*rMsFromLastExec/1000;
		ELSE
			//Define the advance. The minimum advance will be 1. The speed is defined in revs per minute
			rAdvance := IclaSim.Parameters.SpeedFactor * UINT_TO_REAL(Icla.Parameter.Jog.VeloSlow)*rMsFromLastExec/1000;
		END_IF
		rActPosition := rActPosition + rAdvance;
		Icla.Status.iActualPosition := REAL_TO_DINT(rActPosition);
	END_IF

	//Basic Moving Absolute code

	IF ncAbsMov = ncPOS_MOVE THEN
		rSpeed := rSpeed + UINT_TO_REAL(Icla.Parameter.iAcceleration)*rMsFromLastExec/1000;
		rSpeed := MIN(rSpeed, UINT_TO_REAL(Icla.Parameter.MoveAbsolute.Velocity)); //Speed limitation
		rAdvance := IclaSim.Parameters.SpeedFactor * rSpeed *rMsFromLastExec/1000;
		rActPosition := rActPosition + rAdvance;
		Icla.Status.iActualPosition := REAL_TO_DINT(rActPosition);
		Icla.Status.IclaStatus:= AXISILE_MOVE_ABSOLUTE;
		IF Icla.Status.iActualPosition > Icla.Parameter.MoveAbsolute.Position THEN
			//xMovingAbs:=FALSE;
			//xIsMovingAbs:=FALSE;
			Icla.Command.MoveAbsolute:=FALSE;
			ncAbsMov := ncHALT_OK;
			rSpeed := 0;
		END_IF
	END_IF

	IF ncAbsMov = ncNEG_MOVE THEN
		rSpeed := rSpeed + UINT_TO_REAL(Icla.Parameter.iAcceleration)*rMsFromLastExec/1000;
		rSpeed := MIN(rSpeed, UINT_TO_REAL(Icla.Parameter.MoveAbsolute.Velocity)); //Speed limitation
		rAdvance := IclaSim.Parameters.SpeedFactor * rSpeed *rMsFromLastExec/1000;
		rActPosition := rActPosition - rAdvance;
		Icla.Status.iActualPosition := REAL_TO_DINT(rActPosition);
		Icla.Status.IclaStatus:= AXISILE_MOVE_ABSOLUTE;
		IF Icla.Status.iActualPosition < Icla.Parameter.MoveAbsolute.Position THEN
			Icla.Command.MoveAbsolute:=FALSE;
			ncAbsMov := ncHALT_OK;
			rSpeed := 0;
		END_IF
	END_IF

	//Start Absolute movement
	IF EDGEPOS(Icla.Command.MoveAbsolute) THEN
		iAbsoluteMovementOrders := iAbsoluteMovementOrders + 1;
		//Defining starting direction of the movement
		IF Icla.Parameter.MoveAbsolute.Position > Icla.Status.iActualPosition + 1 THEN //Adding safety to avoid loop
			ncAbsMov := ncPOS_MOVE;
		ELSIF Icla.Parameter.MoveAbsolute.Position < Icla.Status.iActualPosition -1 THEN //Adding safety to avoid loop
			ncAbsMov := ncNEG_MOVE;
		ELSE
			Icla.Command.MoveAbsolute:=FALSE;
		END_IF
	END_IF
	IF (ncAbsMov = ncPOS_MOVE OR ncAbsMov = ncNEG_MOVE) AND Icla.Command.Stop THEN
		ncAbsMov := ncHALT_OK;
		Icla.Command.MoveAbsolute:=FALSE;
		Icla.Command.Stop:=FALSE;
		rSpeed := 0;
	END_IF

	//Return the speed depending on the state
	IF Icla.Command.JogForward THEN
		Icla.Status.IclaStatus:= AXISILE_JOG;
		IF Icla.Command.JogFastSpeed THEN
			Icla.Status.iActualVelocity := Icla.Parameter.Jog.VeloFast;
		ELSE
			Icla.Status.iActualVelocity := Icla.Parameter.Jog.VeloSlow;
		END_IF
	ELSIF Icla.Command.JogBackward THEN
		Icla.Status.IclaStatus:= AXISILE_JOG;
		IF Icla.Command.JogFastSpeed THEN
			Icla.Status.iActualVelocity := -Icla.Parameter.Jog.VeloFast;
		ELSE
			Icla.Status.iActualVelocity := -Icla.Parameter.Jog.VeloSlow;
		END_IF
	ELSIF (ncAbsMov = ncPOS_MOVE OR ncAbsMov = ncNEG_MOVE) THEN
		Icla.Status.IclaStatus:= AXISILE_MOVE_ABSOLUTE;
		Icla.Status.iActualVelocity:=Icla.Parameter.MoveAbsolute.Velocity;
	ELSE
		Icla.Status.IclaStatus:= AXISILE_READY;
		Icla.Status.iActualVelocity:=0;
	END_IF

	Icla.Status.xInPosition:= NOT Icla.Command.JogBackward AND NOT Icla.Command.JogForward AND (ncAbsMov = ncHALT_OK);

	Icla.Status.xModuleOK:=TRUE;

	IF Icla.Status.IclaStatus <> AXISILE_ERROR THEN
		Icla.Status.iDriveStatus := ICLAST_ENABLE_OPERATION;
	END_IF

	tiLastExec := clock_ms();

	iIclaSimIndex := iIclaSimIndex + 1;

END_PROGRAM
```

#### IclaSim.var - Local variables
```iecst
VAR
	Icla : REFERENCE TO stIcla;
	IclaSim : REFERENCE TO stIclaSim;
	ncAbsMov : UINT := ncHALT_OK;
	rMsFromLastExec : REAL;
	tiLastExec : TIME;
	rAdvance : REAL;
	rActPosition : REAL;
	rSpeed : REAL;
	iAbsoluteMovementOrders : UINT;
END_VAR
```

### Media Control.md
```markdown
# Media Control

This document explains the media control in the EFI machines. Printer, Dryer and the machines using this ExtPack.

The main scope of this feature is controlling the position and the height of the media inside the machine, considering up to 2 lines in DTP configuration.

With the stack functionality, the machine will be receiving the information of each media before entering the machine, so detailed control of needs can be achieved.

The main functionalities of this Package are:

- Thickness of the blocks

- Activation of Curing (white and color)

- Activation of Drying

- Power of Drying needed

# Notation

`Variable_In_AutomationStudio` or `Method_In_OpcUa`

<mark>Program_In_AutomationStudio</mark>

**Action_In_AutomationStudio**

# Preliminary

Originally, this functionality was just working with arrays, defining the position of the media and the minimum allowed value for the position of the bars. At this point, only the concept of Continuous Media was considered.

The MediaTracking functionality takes the information of the media is entering in the machine and manage the position of each individual media inside the machine. This functionality is need for advance functionalities as DDC (Dynamic Duty Cycle) for Dryer and can be use for Curing and visualization too.

As the need of controlling individual and different media in the printer appeared (mainly for Cube), the NewMediaStack functionality was added. With this functionality, the machine needs to know the media will be entering in the machine. That information will come through an OpcUa Method as `LoadNewMedia` or `LoadNewMediaEnergy`.

<img src=".\.images\summary.png" title="" alt="" data-align="center">

# Program's Architecture

One of the main goals of this feature is consuming as less resources as possible. To achieve it, all the different packages related have been splitted between Fast and Slow programs:

- Fast programs are run with maximum desired speed, so they are defining the maximum information that is managed.

- Slow programs move the information from the Fast programs into the correspondent arrays.

- The result of dividing slow programs Cycle Times between Fast Program Cycle times MUST be an integer and inferior to 10.

  - 4ms and 12ms [3] is allowed

  - 2ms and 10ms [5] is allowed

  - 4ms and 10ms [2.5] is NOT allowed

  - 2ms and 22ms [11] is NOT allowed

## Fast Programs

Fast sensor programs read the information directly form the sensors and store it in their status values.

<mark>ThicknessCtrl_Fast</mark> takes the information from the sensor programs and stores them inside internal arrays for them to be managed later by the slow program.

## Slow Programs

Slow sensor programs manage the non critical and fast information from each type. Homing, slow alarms, communications and others are managed here.

<mark>ThicknessCtrl</mark> is the main program for this functionality. It takes the information from the fast program and moves it into the arrays where the information is treated.

The arrays have a resolution of 1cm, so each position in the array corresponds to 1cm. In the different arrays is stored the presence/absence of some media and the thickness value required for the system.

One key point of the implementation is be receptive to gaps. If the fast program detects a gap, when moving the information to the slow programs, a gap MUST appear, to assure a proper management of the start and the end of each media

## Programs List

The main program is <mark>ThicknessCtrl</mark>. This is the program that collects the data from the different programs, which take the value of the presence and the thickness of the media entering the machine:

- <mark>ThicknessCtrl </mark>[MAIN]

- <mark>nSensorCtrl </mark>[Array of digital sensors with a motor to moving them]

- <mark>AnalogThicknessCtrl </mark>[Analog sensor array]

- <mark>BasicMediaDetect </mark>[Just detecting presence and not thickness of media]

# Basic Operation

The main functionality is running in the <mark>ThicknessCtrl</mark> program. This is the main Slow program of the package.

When the Belt is running and the speed is higher than minimum, the program calculates the `iPositionsToRunArray`. This is a key point in the program. The centimeters that the arrays has to be moved, considering the speed of the belt and the program cycle.

If  `iPositionsToRunArray > 0`, then the program moves the arrays to consider the new desired position of the data. The arrays are shifted with the function `ShiftArrayForward` a certain number of positions determined by `iPositionstoRunArray`. This action moves all the elements towards the end of the array that number of positions.

- **RunHeightArray** manages the thickness of the media with `iHeightArray`

- **RunMediaArray** manages the presence of media with `xMediaTracking`

<img title="" src="./.images/shiftArrayFW.png" alt="" width="114" data-align="center">

## RunHeightArray

This Action moves the information in  `iHeightArray` and loads the height from the sensor information depending on the system installed in the machine.

After moving/shifting and loading new data, the maximum thickness per each enabled section is calculated. Each section is used by one block to define the minimum position the block can be positioned.

### Sections

Sections are defined for when a machine has more than one block or area. This way, the height can be controlled independently for each one of them. Each section would be updated with the minimum vertical position needed to avoid crash.

## RunMediaArray

This Action shifts the information inside `xMediaTracking`, then filters, checks and loads the new values from the source of the media inside this array.

`xMediaTracking` will then contain information of the presence of media all along the distance  considered in each machine.

Media data presence is filtered to avoid false positives (ink in the belt) and it is checked for consistency

## Position Array

The ***PositionArray*** file is an aggrupation of functions that recalculate distances to adjust them to the current position of the pieces taking into account `iPositionToRunArray`, which is the distance that the pieces move within a cycle period, and it is calculated in function of the belt speed and the cycle period.

The feature works in one centimeter steps, but yet the distance can take a non-integer value. So between cycles, the distance gained can have some decimals to it. Those extra distances cannot be directly added and are instead added up to a buffer and only when that addition exceeds the unit, the integer part is added for compensation.

# Media Tracking

This functionality consists in tracking the pieces that pass through the machine, taking account of the presence and absence of pieces to identify gaps and differentiate pieces between them.

`xMediaTracking` is the array over this functionality operates and the process is as follows:

This function detects whenever a piece enters the machine, and also calculates the number of pieces inside.

The information tracked by the functionality is the media data (thickness, dimensions, white, energy, etc.) plus the important information for tracking. This information is stores in `MediaTrackingInsideL1 `and `MediaTrackingInsideL2`.

- `HeadPosition` for tracking the position head of the media and and managing functions like curing activation timing and drying.

- `TailPosition` for tracking the tail position of the media. A `TailPosition = 0` is considered a media still entering in the machine.

<img title="" src=".images/shiftArrayBW.png" alt="" data-align="center" width="436">

In case either the Curing or Drying functionalities are enabled in MediaTracking, it will also take into account inside positions and check for exiting media.

## CureTracking

***CureTracking*** contains functions for activating  the curing lamps only if one piece is under the lamps.

When *MediaControl* is enabled, the program will have the curing lamps on when any portion of a piece is under the curing window. This is a diagram explaining the possible states of a piece in relation to the curing lamps (*Curing Window*) and the state of the lamps.

![](.\.images\curingWindow.png)

- On **State A** the piece has not arrived to the curing yet. So the lamps will be **OFF**

- On **States labeled with a B**, where there is a piece below he Curing Window (in the case of **B.1** it is only the head, in the case of **B.3** it is only the tail, but that does not matter), so the lamps must be **ON**

- On **State C**, the whole piece has exited the area below the Curing Window, so the leds can be set **OFF** again.

## DryTracking

The DryTracking functionality is an extra functionality of the MediaTracking. When it is activated, besides to the media itself, it is received the information of the Energy needed to Dry the media. This information can come from the Stack functionality or from the ContinuousMedia structure.

### With Stack Functionality

When Stack is activated, the Energy information is place in the `MediaEnergyRackL1`  or `MediaEnergyRackL2` when loaded the information to the Stack.

When the media enters in the machine, the Media is assigned to MediaTrackingInsideL1 with the media itself and the pointer to the Energy information.

### Without Stack. Continuous Media

When Stack is NOT activated, the Energy information is place in the `MediaEnergyRackL1` or `MediaEnergyRackL2` from `ContinuousMedia.Energy` when entering media to the machine

# New Stack Media

This feature operates by the principle of a FIFO (First In First Out) queue, which means that the first piece to enter the queue is the first one to be treated.
Press Software supplies data about the media that will be entering the machine, which are then stored inside an array along all the other data necessary when the media enters the machine.

Some of the more important parameters are:

- **Thickness**: for the machine to adjust the height of the bars.
- Need of **white Ink** depending on whether the piece needs it or not, the **curing LEDs** for white will need to turn on or not, this way having them on all the time can be avoided.

This functionality is implemented in the action **MediaTracking**.  The main actions inside this main action are:

* **CheckFinishEnteringMedia**: Review end of media currently entering. Assign `TailPosition`

* **CheckEnteringMedia**: Review  start of the media. Assign `HeadPosition`

* **RunMediaInsidePositions**; Increase the values of `HeadPosition `and `TailPosition`

* **CheckExitingMedia**: Review the media exiting of the machine

### Moving elements between arrays

When some new media enters (if stack is enabled for detection) the first item from the `NewMediaStackLX` array has to be moved into the last position of `InsideMediaStackLX`. When doing so, the first position remains empty, so all the elements inside `NewMediaStackLX` have to be shifted towards the beginning of the array.

This is done with the `ShiftArrayBackward` action, that moves all the elements inside an array towards the beginning.

<img title="" src=".images/shiftArrayBW.png" alt="" data-align="inline" width="436">

## Reject tracking

The feature also track rejected pieces. It stores the *validity* of the pieces inside another array called `ValidMedia`.

## Alarms

Mainly, there is one new alarm defined: *"NoThicknessInstalled"*, which detects if, for any reason and while having the proper sensors on the machine, there is no information about the thickness of a piece. This alarm will stop the machine.
```

### Program Logical/ExtPack/_Media/AnalogThicknessCtrl/AnalogThicknessCtrl_v1/AnalogThickness (IEC)

#### Alarms.st
```iecst
ACTION alarms:

	//////////////////////////
	//ALARMS
	//////////////////////////

	// Alarm: Incoherence Ding detect

	// Alarm: Fault Ding detection signal, it comes from mapping inputs
	data.Alarms.xAlNoDingDetect:=data.In.xDingChannelFault OR NOT data.In.xModuleOK;

	// Alarm: Ding is not referenced-
	data.Alarms.xAlDingNotReferenced:= NOT data.State.xDingReferenced;

	// Reference issue CRETALEGO-909/911: Alarm: tile thickness read too low after bars is positioned in print.
	data.Alarms.xAlDingIncoherenceValue:= gBelt.states.xRuningBelt AND (data.State.rCurrentHigh < data.Parameters.rMachineMinTicknessMedia) AND EDGEPOS (data.In.xAnyCarriageProductDetect) AND data.In.xDingLow;

	// Alarm: No digital Ding Detect
	T_NoDigDingDetect.IN:= (data.State.rCurrentHigh < data.Parameters.rMachineMinTicknessMedia) AND data.In.xDingLow AND NOT data.In.xDingChannelFault;
	T_NoDigDingDetect.PT:= T#200ms;
	T_NoDigDingDetect();

	// TILE THICKNESS READ  IS TOO LOW. CHECK THE SETTINGS OF THE TILE DETECTION LASER.
	IF T_NoDigDingDetect.Q OR data.Alarms.xAlDingIncoherenceValue THEN
		data.Alarms.xAlDingNoDigLaserSensor:= TRUE;
	END_IF

END_ACTION
```

#### AlarmSounds.st
```iecst
ACTION AlarmSounds:

	ars_AlMountedTile.xAlarm:= data.Alarms.xMountedTile;
	ars_AlMountedTile.xSilence:= data.Commands.xMute;
	ars_AlMountedTile();

	ars_AlDingConexionError.xAlarm:= data.Alarms.xAlDingConexionError;
	ars_AlDingConexionError.xSilence:= data.Commands.xMute;
	ars_AlDingConexionError();

	ars_AlDingNotReferenced.xAlarm:= data.Alarms.xAlDingNotReferenced;
	ars_AlDingNotReferenced.xSilence:= data.Commands.xMute;
	ars_AlDingNotReferenced();

	ars_AlNoDingDetect.xAlarm:= data.Alarms.xAlNoDingDetect;
	ars_AlNoDingDetect.xSilence:= data.Commands.xMute;
	ars_AlNoDingDetect();

	ars_AlDingDetect.xAlarm:= data.Alarms.xAlDingDetect;
	ars_AlDingDetect.xSilence:= data.Commands.xMute;
	ars_AlDingDetect();

	ars_AlDingIncoherenceValue.xAlarm:= data.Alarms.xAlDingIncoherenceValue;
	ars_AlDingIncoherenceValue.xSilence:= data.Commands.xMute;
	ars_AlDingIncoherenceValue();

	ars_AlDingNoDigLaserSensor.xAlarm:= data.Alarms.xAlDingNoDigLaserSensor;
	ars_AlDingNoDigLaserSensor.xSilence:= data.Commands.xMute;
	ars_AlDingNoDigLaserSensor();

	data.AlSummary.xAlarmSound:=	ars_AlDingConexionError.xAlarmSound OR
									ars_AlDingNotReferenced.xAlarmSound OR
									ars_AlNoDingDetect.xAlarmSound OR
									ars_AlDingDetect.xAlarmSound OR
									ars_AlDingIncoherenceValue.xAlarmSound OR
									ars_AlDingNoDigLaserSensor.xAlarmSound OR
									ars_AlMountedTile.xAlarmSound;

END_ACTION
```

#### AnalogThickness.st
```iecst
PROGRAM _CYCLIC

	//Main data assignation
	data ACCESS ADR (gDing);

	// Assigning status.xInstalled considering dynamic enable
	IF data.Parameters.xDingInstalled THEN
		IF data.Parameters.xAllowDynamicEnable THEN
			data.State.xDingInstalled:= data.Parameters.xEnable;
		ELSE
			data.State.xDingInstalled:= TRUE;
		END_IF
	ELSE
		data.State.xDingInstalled:= FALSE;
	END_IF

	//If not installed, clear alarms and exit
	IF NOT data.State.xDingInstalled THEN
		ResetAlarms;
		ResetCommands;
		data.State.xDingReferenced:=FALSE;
		RETURN;
	END_IF

	// Checking values
	gDing._Internal.rMarginSafePrintChecked := MAX(gDing.Parameters.rMarginSafePrint, 1.0); //The minimum Margin Safe print is 1mm

	// Recovering calibration data if configured
	IF data.State.xDingInstalled AND data.Parameters.xKeepHoming AND NOT xRecoveredPermanentInfo THEN
		data.State.xDingReferenced := data.State.Permanent.xDingReferenced;
		data.State.rOffsetCalibration := data.State.Permanent.rOffsetCalibration;
		xRecoveredPermanentInfo := TRUE;
	END_IF

	//Reset Alarms with the reset command
	IF data.Commands.xErrorRst THEN
		ResetAlarms;
	END_IF

	//With Zero and the command to calibrate, the system is not calibrated
	IF data.Commands.Mode.xZero AND data.Commands.xCalibrateThickness THEN

		data.State.xDingReferenced:=FALSE;

		IF data.In.xDingLow THEN
			LogOrderReceivedOK;

			IF ABS(data.parSw.rCalibrationValue-data.In.rHighDingMm) < 3.0 THEN
				data.State.rOffsetCalibration:=data.parSw.rCalibrationValue-data.In.rHighDingMm;
				data.State.xDingReferenced:=TRUE;
				data.Alarms.xAlDingNoMediaToCalibrate:=FALSE;
				LogCalibrationOK;
			END_IF

		ELSE
			//If Order to calibrate and not media in the sensor, raise a Warning Alarm
			data.Alarms.xAlDingNoMediaToCalibrate:=TRUE;
			LogOrderReceivedNOK;
		END_IF

	END_IF

	//Take the command as an edge
	IF data.Commands.xCalibrateThickness THEN
		data.Commands.xCalibrateThickness:=FALSE;
	END_IF

	// NOTE: Keep this code until check in machine the efectiveness of the next code to avoid running through an array
	//	arrThickness[0]:=REAL_TO_INT(data.State.rCurrentHigh*10.0);
	//	iMaxThicknessToSw:=0;
	//	FOR iIndexThickness:=VALUES_TO_GET_MAX_THICKNESS TO 1 BY -1 DO
	//		arrThickness[iIndexThickness]:= arrThickness[iIndexThickness-1];
	//		iMaxThicknessToSw:=MAX(iMaxThicknessToSw, arrThickness[iIndexThickness]);
	//	END_FOR;
	//	data.State.rCurrentThicknessStable:=INT_TO_REAL(iMaxThicknessToSw)/10.0;

	RTC_gettime(ADR(timeReaded));
	iModSec := timeReaded.second MOD 3;
	IF EDGEPOS(iModSec=0) THEN rMaxThicknessS0:=0; END_IF
	IF EDGEPOS(iModSec=1) THEN rMaxThicknessS1:=0; END_IF
	IF EDGEPOS(iModSec=2) THEN rMaxThicknessS2:=0; END_IF
	rMaxThicknessS0 := MAX(rMaxThicknessS0, data.State.rCurrentHigh);
	rMaxThicknessS1 := MAX(rMaxThicknessS1, data.State.rCurrentHigh);
	rMaxThicknessS2 := MAX(rMaxThicknessS2, data.State.rCurrentHigh);
	rMaxThickness := MAX(rMaxThicknessS0, rMaxThicknessS1, rMaxThicknessS2);
	data.State.rCurrentThicknessStable:=rMaxThickness;

	// Counter of Dinf low piece detect
	IF EDGEPOS (data.State.xDingLowPieceDetect) THEN
		data.State.diLgLowPieceCounter:= data.State.diLgLowPieceCounter+1;
	END_IF;

	///////////////
	//ALARMS
	//////////////
	alarms;

	AlarmsSummary;

	AlarmSounds;

	data.Out.xReset := data.In.xDingChannelFault AND data.Commands.xErrorRst;

	// Storing current data in permanent
	data.State.Permanent.rOffsetCalibration := data.State.rOffsetCalibration;
	data.State.Permanent.xDingReferenced := data.State.xDingReferenced;

	///////////////////////////
	// Mounted media management. ThicknessCtrl MUST be executed in the slow cycle before this program
	IF data.State.xMountedMediaDetected AND NOT data._Internal.xMountedMediaTreated THEN
		data._Internal.xMountedMediaTreated := TRUE;
	END_IF
	IF NOT data.State.xMountedMediaDetected THEN
		data._Internal.xMountedMediaTreated := FALSE;
	END_IF

	///////////////////////////
	// Media To Reject management. ThicknessCtrl MUST be executed in the slow cycle before this program
	IF data.State.xMediaToRejectDetected AND NOT data._Internal.xMediaToRejectTreated THEN
		data._Internal.xMediaToRejectTreated := TRUE;
		LogRejectDetected;
	END_IF
	IF NOT data.State.xMediaToRejectDetected THEN
		data._Internal.xMediaToRejectTreated := FALSE;
	END_IF
	IF EDGENEG(data.State.xMediaToRejectDetected) THEN
		LogRejectEnded;
	END_IF

END_PROGRAM
```

#### EventLog.st
```iecst
ACTION LogOrderReceivedOK:
	stEventLog.Source := ELOG_TYPE_DETECTION;
	stEventLog.Severity:= ELOG_SEVERITY_INFO;
	stEventLog.Facility:= 0;
	stEventLog.ErrorCode:=0;
	stEventLog.Text := 'Analog Thickness sensor order received';
	gEventLogLoader(EventData := ADR(stEventLog));
END_ACTION

ACTION LogOrderReceivedNOK:
	stEventLog.Source := ELOG_TYPE_DETECTION;
	stEventLog.Severity:= ELOG_SEVERITY_INFO;
	stEventLog.Facility:= 0;
	stEventLog.ErrorCode:=0;
	stEventLog.Text := 'Analog Thickness sensor order received but not Media in sensor. Action cancelled';
	gEventLogLoader(EventData:=ADR(stEventLog));
END_ACTION

ACTION LogCalibrationOK:
	stEventLogCal.Source := ELOG_TYPE_DETECTION;
	stEventLogCal.Severity:= ELOG_SEVERITY_INFO;
	stEventLogCal.Facility:= 0;
	stEventLogCal.ErrorCode:=0;
	stEventLogCal.Text := 'Analog Thickness sensor calibrated with offset: ';
	brsftoa(gDing.State.rOffsetCalibration, ADR(strAux));
	brsstrcat(ADR(stEventLogCal.Text), ADR(strAux));
	brsstrcat(ADR(stEventLogCal.Text), ADR('mm'));
	gEventLogLoader(EventData:=ADR(stEventLogCal));
END_ACTION

ACTION LogRejectDetected:
	stEventLogReject.Source := ELOG_TYPE_DETECTION;
	stEventLogReject.Severity:= ELOG_SEVERITY_INFO;
	stEventLogReject.Facility:= 0;
	stEventLogReject.ErrorCode:=0;
	stEventLogReject.Text := 'Analog. Rejected Media Detected';
	gEventLogLoader(EventData := ADR(stEventLogReject));
END_ACTION

ACTION LogRejectEnded:
	stEventLogEndReject.Source := ELOG_TYPE_DETECTION;
	stEventLogEndReject.Severity:= ELOG_SEVERITY_INFO;
	stEventLogEndReject.Facility:= 0;
	stEventLogEndReject.ErrorCode:=0;
	stEventLogEndReject.Text := 'Analog. End Rejected Media Detection';
	gEventLogLoader(EventData := ADR(stEventLogEndReject));
END_ACTION
```

### Program Logical/ExtPack/_Media/AnalogThicknessCtrl/AnalogThicknessCtrl_v1/Analog_Fast (IEC)

#### InAnalogThickness.var
```iecst
VAR
	dingCard : REFERENCE TO PlcCardMapping;
	rThicknessToMounted : REAL;
	xMountedMediaDetected : BOOL;
	xMediaToRejectDetected : BOOL;
	iMaxSamples : USINT;
	iHighDingRaw : INT;
	iIndexSamples : USINT;
	rVirtualDiscretePosition : REAL;
	rBarsPosition : REAL;
	iIndexVirtualSensor : USINT;
END_VAR
```

### Program Logical/ExtPack/_Media/BasicDetectMediaCtrl/BasicDetectMediaCtrl_v1/BasicDetectMediaCtrl (IEC)

#### DetectionMediaCtrl.st - Cyclic code
```iecst
PROGRAM _INIT

	vData ACCESS ADR(gBasicDetectMedia);
	vData.Parameters.rDesiredHeigh := 20;

END_PROGRAM

PROGRAM _CYCLIC

	vData ACCESS ADR(gBasicDetectMedia);

	IF NOT vData.Parameters.xInstalled THEN
		vData.Status := StatusReseted;
		RETURN;
	END_IF

	IF vData.Commands.xReset THEN
		vData.Alarms := AlarmsReseted;
	END_IF

	vData.Status.xInstalled := vData.Parameters.xInstalled;
	vData.Status.xMediaPresent := vData.Inputs.xMediaPresentL1 OR vData.Inputs.xMediaPresentL2;

	//Define Alarms
	IF vData.Inputs.xMountedMedia AND vData.Parameters.xBeltMoving THEN
		vData.Alarms.xMountedMedia := TRUE;
	END_IF

	IF vData.Inputs.xCorrection THEN
		vData.Status.rMediaHeigh := vData.Parameters.rDesiredHeigh + vData.Parameters.rCorrection;
	ELSE
		vData.Status.rMediaHeigh := vData.Parameters.rDesiredHeigh;
	END_IF

	//Sound managing
	arMountedMedia		(xAlarm:= gDryer.Al.Alarm.xAlarmMountedMedia, xSilence:=gDryer.AutoCmd.xMuteAlarms);

	iReasonSound.0 := arMountedMedia.xAlarmSound;
	vData.AlSummary.xAlarmSound := iReasonSound > 0;

END_PROGRAM
```

#### DetectionMediaCtrl.var - Local variables
```iecst
VAR
	vData : REFERENCE TO DetectionMedia;
	StatusReseted : DetectionMedia_Status;
	AlarmsReseted : DetectionMedia_Alarms;
	arMountedMedia : AutoResetSound;
	iReasonSound : UINT;
END_VAR
```

### nSensorCtrl.typ
```iecst
TYPE
	nSensors_typ : 	STRUCT
		ordersSw : nSensorsOrdersSw; (*Orders from sw*)
		commandsSw : nSensorsCommandsSw; (*Commands gui*)
		commands : nSensorsCommands; (*Commands gui*)
		parameters : nSensorsParameters; (*Parameters gui*)
		parSw : nSensorsParametersSw;
		status : nSensorsStatus; (*States potocell system*)
		Alarms : nSensorsAlarms; (*Alarms*)
		AlSummary : stEFI_AlarmSummary; (*Alarms Summary*)
		Inputs : nSensorsInputs;
		_Internal : nSensorsInternal;
	END_STRUCT;
	nSensorsOrdersSw : 	STRUCT
		xMoveUp : BOOL;
		xMoveDown : BOOL;
	END_STRUCT;
	nSensorsCommandsSw : 	STRUCT
		xReference : BOOL;
	END_STRUCT;
	nSensorsCommands : 	STRUCT
		xOrderQuickStop : BOOL;
		xOrderCap : BOOL;
		xErrorRst : BOOL;
		xMute : BOOL;
		xRecordMaxPosition : BOOL; (*To save bars position only when this command is active*)
		xCheckMounted : BOOL;
		xCancelAlignmentCheck : BOOL;
		AutoMode : stEFI_MachineAutoModes;
		Mode : StGeneral_States_Mode;
		xResetMotor : BOOL;
		LineStatusSummary : LineControlStatusSummarized;
		xMountedMediaInside : BOOL; (*Mounted Media inside*)
		xStartCount : BOOL;
	END_STRUCT;
	nSensorsSensorParSw : 	STRUCT
		xToRejectMedia : BOOL; (*The sensor marks media to be rejected due to low printing quality once bars will move up due to its detection*)
	END_STRUCT;
	nSensorsSensorParameters : 	STRUCT
		rSafetyOffset : REAL;
		rDistanceRelativeToFirstSensor : REAL; (*Distance between Sensor and first sensor in mm*)
		rDistanceToBase : REAL; (*Distance to belt surface*)
		xMountedMedia : BOOL; (*The sensor actives mounted media alarm*)
		xEnabled : BOOL; (*The sensor changes print bar position to next photocell's position*)
		xMoveBarsUp : BOOL; (*The sensor changes print bar position to next photocell's position*)
	END_STRUCT;
	nSensorsParametersSw : 	STRUCT
		rMechOffset : REAL := 0.0; (*Offset in mm*)
		rThicknessReference : REAL := 10; (*Thickness of the media while referencing in mm*)
		Sensors : ARRAY[0..MAX_LAST_NSENSOR]OF nSensorsSensorParSw; (*Sensors 0 and 1 invalid. Using from 2 to limit*)
	END_STRUCT;
	nSensorsParameters : 	STRUCT
		xInstall : BOOL;
		xEnable : BOOL; (*Configured depending on the machine. Is installed or it can be installed*)
		xAllowDynamicEnable : BOOL; (*The machine allows dynamic enabling or disabling the funcionality*)
		MotorType : nSensorsMotorsType;
		DriveUnit : MC_DriveUnitManager;
		Sensors : ARRAY[0..MAX_LAST_NSENSOR]OF nSensorsSensorParameters; (*Sensors 0 and 1 invalid. Using from 2 to limit*)
		AlignmentProcess : nSensorsAlignmentProcess;
		IndexDriveMaster : USINT; (*Index of the primary (master) motor in gAxis array*)
		IndexDriveSecondary : USINT; (*Index of the secondary (gear) motor in gAxis array*)
		iSensorQuantity : USINT; (*Quantity of the sensors used*)
		IndexIcla : USINT; (*Index of the Icla in Icla array*)
		iSensorToReference : USINT; (*Sensor to define the position at homing*)
		rSensorMechToleranceAlignment : REAL := 5; (*Teorical alignment position tolerance as mechanical specification*)
		rSensorTeoMechPositionAlignment : REAL; (*Teorical alignment position as mechanical specification*)
		rSensorMechPositionAlignmentMin : REAL; (*Minimum alignment position allowed*)
		rSensorMechPositionAlignmentMax : REAL; (*Maximum alignment position allowed*)
		rSensorMechPositionMin : REAL := -3; (*Mechanical max position allowed is -15mm. Value get from Andres Mantilla after reviewing nSensor mechanical assembly*)
		rSensorMechPositionMax : REAL := 75; (*Mechanical max position allowed*)
		rSensorPositionSearchAlignment : REAL := 50; (*Position to avoid false gauge detections*)
		rOffsetRelToBar : REAL := 0.0; (*Media Offset position in mm. Distance to position third or fourth laser below the print bar. Testing purposes DELOREAN-2572*)
		rOffsetPosition : REAL := 0.0; (*Media Offset position in mm. The offset in position to placed the sensors*)
		rMarginPrint : REAL; (*Value in mm*)
		rMediaThickness : REAL := 5; (*Media Thickness in mm*)
		Acceleration : REAL := 500; (*Acc SP mm/ s2*)
		JogSpeed : REAL := 10; (*Jog Speed SP mm/s*)
		Speed : REAL := 100; (*Speed SP mm/s*)
		rDistanceBetweenSensors : REAL; (*Distance between Sensors in mm*)
		rSensorMechPositionByPass : REAL := 50; (*Static position for ByPass mode*)
		xEnableMountedAlrByPass : BOOL; (*Enable Mounted Part In By Pass Mode*)
		xSensorsPosHybridBehaviour : BOOL;
		xRaiseMountedJustBelowPrePrint : BOOL; (*The RaiseMounted alarm is just raised if Motor Below PrePrintPosition*)
		rPrePrintPosition : REAL; (*PrePrintPosition of the first block*)
		xHomingEnabled : BOOL; (*Transvacuums are activated. Used to start homing movements*)
	END_STRUCT;
	nSensorsStatus : 	STRUCT
		iErrorId : UINT;
		xMotorError : BOOL;
		xInstalled : BOOL;
		xReferencing : BOOL;
		xReferenced : BOOL;
		xFrontModuleOk : BOOL;
		xBackModuleOk : BOOL;
		xAllPhotoInactive : BOOL;
		xSensorsSeparatedInProcessDir : BOOL; (*Active when photocell are not assemble over the same vertical axis. That means there is a distance<>0  between them in process direction*)
		xTrustPhotocellASignal : BOOL; (*Active when photocell is over the belt and its signal can be trusted*)
		iSystemState : nSensorsStateMotors := STP_NOT_INITIALIZED;
		iBlocksPositionDesired : INT;
		rSensorPositionAlignment : REAL; (*Position of motor to check alignment of sensors*)
		rBarsPosition : REAL; (*Minimum position of the bar to avoid a crash. Value in mm*)
		rPositionWithOffset : REAL; (*Position in mm of the motors considering the offset. This is equal to the MediaThickness set point*)
		rPositionMotor : REAL; (*Position in mm of the motors*)
		rOffsetToReject : REAL; (*Position to reject the media. Just the second sensor from top*)
		rOffsetToMounted : REAL; (*Position to consider mounted media. Just the first sensor from top*)
		rOffsetToApplyToBarsPosition : REAL;
		xSensorsPositionedRelativeToBar : BOOL; (*Variable to define position desired mode*)
		iSensorToApplyOffset : USINT; (*Index of sensor used to be positioned below bars a distance = rOffsetRelToBar*)
		xInPosition : BOOL; (*Sensors are in the right position depending on the media thickness*)
		xBelowSetPoint : BOOL; (*Sensors are Below the right position depending on the media thickness*)
		xAboveSetPoint : BOOL; (*Sensors are Above the right position depending on the media thickness*)
		xAlignmentChecked : BOOL;
		xCheckingAlignment : BOOL; (*TRUE if in any of the states checking alignement*)
		xSensorValidAlignPos : BOOL;
		xLowPieceDetect : BOOL; (*Low Sensor Detectect*)
		iDetectCount : ARRAY[0..MAX_LAST_NSENSOR]OF UINT; (*Variable to save number of detetions of each sensor*)
		xPhotoCellsNotAligned : ARRAY[0..MAX_LAST_NSENSOR]OF BOOL; (*Signal is TRUE when photocell is not aligned*)
		xMediaToRejectDetected : BOOL; (*Media to be rejected has beed detected*)
		xMountedMediaDetected : BOOL; (*Mounted media has been detected*)
		Icla : nSensors_IclaStatus;
	END_STRUCT;
	nSensorsAlarms : 	STRUCT
		xNotReferenced : BOOL; (*Phocell system not homed*)
		xNotInstalled : BOOL;
		xComsMotorError : BOOL;
		xMountedTile : BOOL; (*Sensor configured as Mounted Media activated*)
		xControllerNotReady : BOOL; (*Waiting for enable input (STO_A, STO_B)*)
		xMotorError : BOOL; (*Error Id != 0*)
		xNoDigSignalLaserSensor : BOOL; (*Pending to remove in 4.3.6*)
		xContinuousActPDPhcell : BOOL; (*Pending to remove in 4.3.6*)
		xIncoherPhotocellSystem : BOOL; (*Pending to remove in 4.3.6*)
		xAlrCriticalPhotocellNotAligned : BOOL; (*There is an operative photocell not aligned*)
		xPositionOutOfRange : BOOL; (*Maximum sensor position allowed*)
		xAlrWarpMedia : BOOL;
		xAlrInvalidAlignmentPosition : BOOL; (*Alignment position is out of allowed range*)
		xPhotoCellsNotAlignedWarning : ARRAY[0..MAX_LAST_NSENSOR]OF BOOL; (*Warning, not operative photocell*)
		xPhotoCellsNotAlignedError : ARRAY[0..MAX_LAST_NSENSOR]OF BOOL; (*Critical, operative photocell*)
		xPhotoCellsDetectionIncoherence : ARRAY[0..MAX_LAST_NSENSOR]OF BOOL; (*Critical, operative photocell*)
	END_STRUCT;
	nSensorsSignalsIn : 	STRUCT
		xPhotoCells : ARRAY[0..MAX_LAST_NSENSOR]OF BOOL; (*Signal 0 not valid. Needed for definition. Starts with 1. This cannot be assigned in mapping. It is intenally assign with the pointers. SOMETHING CROSSING, value 0*)
		pInput : ARRAY[0..MAX_LAST_NSENSOR]OF UDINT; (*Pointers to the input card of the photocells signal*)
		xSafetyEnable : BOOL;
	END_STRUCT;
	nSensorsStateMotors :
		(
		STP_NOT_USED,
		STP_NOT_INITIALIZED,
		STP_POWER_ON,
		STP_HOME_DIR,
		STP_GEARING,
		STP_GEARED,
		STP_HOMING_STEP_1,
		STP_HOMING_STEP_2,
		STP_HOMING_STEP_3,
		STP_HOMING_STEP_4,
		STP_SEARCH_ALIGNMENT_POS_STEP_1,
		STP_SEARCH_ALIGNMENT_POS_STEP_2,
		STP_SEARCH_ALIGNMENT_POS_STEP_3,
		STP_SEARCH_ALIGNMENT_POS_STEP_4,
		STP_CHECK_ALIGNMENT_STEP_1,
		STP_CHECK_ALIGNMENT_STEP_2,
		STP_CHECK_ALIGNMENT_STEP_3,
		STP_CHECK_ALIGNMENT_STEP_4,
		STP_CHECK_ALIGNMENT_STEP_5,
		STP_CHECK_ALIGNMENT_STEP_6,
		STP_STANDSTILL,
		STP_JOGGING,
		STP_AUTO,
		STP_SET_POS,
		STP_RUNING,
		STP_ERROR
		);
	nSensorsAlignmentProcess :
		(
		STP_ALIGNMENT_NO_REQUIRED,
		STP_ALIGNMENT_REQUIRED
		);
	nSensorsMotorsType :
		(
		STP_STEPPER,
		STP_ICLA
		);
	nSensorsInputs : 	STRUCT
		Signals : nSensorsSignalsIn; (*Signal 0 not valid. Needed for definition. Starts with 1*)
	END_STRUCT;
	nSensorsInternal : 	STRUCT
		xMediaToRejectTreated : BOOL; (*Media to Reject has been treated and can be reseted if the sensor is not detecting*)
		xMountedMediaTreated : BOOL; (*Mounted media has been treated and can be reseted if the sensor is not detecting*)
		rMarginSafePrintChecked : REAL; (*Fix offset to bent tile. The heads go to the thickness measured + this value. Value in mm. Checked minimum value*)
	END_STRUCT;
	nSensors_IclaStatus : 	STRUCT
		iIclaState : INT; (*Drive status state machine Icla*)
		xHomed : BOOL;
		xIsMoving : BOOL;
		xHoming : BOOL;
		rCurrentVel : REAL; (*Current position in mm*)
		rMaxTorque : REAL; (*Current position in mm*)
		rCurrentTorque : REAL; (*Current position in mm*)
		rCurrentPosition : REAL; (*Current position in mm*)
		iErrorId : UINT;
	END_STRUCT;
END_TYPE
```

### Program Logical/ExtPack/_Media/nSensorCtrl/nSensorCtrl_v2/nSensorCtrl

#### nSensorCtrl.var
```iecst
VAR
	data : REFERENCE TO nSensors_typ;
	stnSensorsAlarmsReseted : nSensorsAlarms;
	stnSensorsAlarmSummaryReseted : stEFI_AlarmSummary;
	Stepper : REFERENCE TO AxisCtrl_typ;
	StepperGear : REFERENCE TO AxisCtrl_typ;
	Icla : REFERENCE TO stIcla;
	rSensorPositionAlignment : REAL; (*Pulses*)
	rSensorPositionAlignmentMax : REAL; (*Pulses*)
	rSensorPositionAlignmentMin : REAL; (*Pulses*)
	rSensorPositionDesired : REAL; (*Pulses*)
END_VAR
VAR CONSTANT
	iHistoryLines : USINT := 20;
END_VAR
VAR
	tonAlignmentProcess : TON;
	tonTimeOutGearing : TON;
	tonMaxTimeJogging : TON;
	xAnyManualMovement : BOOL;
	xAnyErrorStepper : BOOL;
	rPositionMotorMm : REAL;
	ars_ComsMotorError : AutoResetSound;
	ars_NotReferenced : AutoResetSound;
	ars_IncoherPhotocellSystem : AutoResetSound;
	ars_InvalidAlignmentPosition : AutoResetSound;
	ars_CriticalPhotocellNotAligned : AutoResetSound;
	ars_MotorError : AutoResetSound;
	iReasonWarning : UDINT;
	iReasonStop : UDINT;
	iReasonCritical : UDINT;
	StateHistory : ARRAY[0..iHistoryLines] OF nSensorsStateMotors;
	iIndexHistory : USINT;
	MotorDriveUnit : DriveUnitMngr;
	rJogSpeedSetPoint : REAL;
	TON_DelayIncoherrPhotocell : TON; (*Delay_Incoher PhotoCell System Alarm*)
	xControllerReady : BOOL;
	xPoweredOn : BOOL;
	xMotorReady : BOOL;
	xAnyManualOrder : BOOL;
	iIndexSensor : USINT;
	xAllSensorInactive : BOOL;
	xAlignmentPositionSet : BOOL;
	xAllSensorActive : BOOL;
	IncoherenceSensor : UINT;
	iAnyAlarm : UINT;
	iAnyWarning : UINT;
	iLastStateToCheckPosition : USINT;
	iStateToCheckPosition : USINT;
	tonMotorStopped : TON;
	xMotorStopped : BOOL;
	xMotorChanged : BOOL;
	PreviousMotorType : nSensorsMotorsType;
	stCriticalAlarmsLog : EventLog_typ;
	stStopAlarmsLog : EventLog_typ;
	stWarningAlarmsLog : EventLog_typ;
	xWarpSensorActive : BOOL;
	xWarpMediaPresent : BOOL; (*Warp media*)
	iWarpMediaSensor : UINT; (*Sensor defined as warp sensor*)
	iCounterWarpMedia : UINT; (*Warp media counter*)
	iMaxWarpMedia : UINT := 2; (*Number of warp boards to raise warp media alarm*)
	TON_ContinuousActPDPhcell : TON;
	arsContinuousActPDPhcell : AutoResetSound;
	iReasonCheckingAlignment : UINT;
	iIndexSensorToPositionBelowBars : USINT;
	rOffsetPositionCalc : REAL;
	rOffsetPosition : REAL;
	xSensorsPositionedRelativeToBar : BOOL;
	xPhotoInputsPrev : ARRAY[0..MAX_LAST_NSENSOR] OF BOOL; (*Previous value of the photocells to allow EDGEPOS in a FOR*)
	ResetCommandsSw : nSensorsCommandsSw;
END_VAR
```

#### EventLog.st
```iecst
ACTION LogWarningAlarm:

	stWarningAlarmsLog.Source := ELOG_TYPE_DETECTION;
	stWarningAlarmsLog.Severity:= ELOG_SEVERITY_INFO;
	stWarningAlarmsLog.Facility:= 0;
	stWarningAlarmsLog.ErrorCode:=0;

	stWarningAlarmsLog.Text := 'nSensorWarningAlarm';

	IF iReasonWarning.0 THEN stWarningAlarmsLog.Text := 'data.Alarms.xReferencing';
	ELSIF iReasonWarning.1 THEN	stWarningAlarmsLog.Text := 'data.Alarms.xNotReferenced';
	ELSIF iReasonWarning.2 THEN	stWarningAlarmsLog.Text := 'data.Alarms.xAlrWarpMedia';
	END_IF

	gEventLogLoader(EventData := ADR(stWarningAlarmsLog));

END_ACTION

ACTION LogStopAlarm:

	stStopAlarmsLog.Source := ELOG_TYPE_DETECTION;
	stStopAlarmsLog.Severity:= ELOG_SEVERITY_INFO;
	stStopAlarmsLog.Facility:= 0;
	stStopAlarmsLog.ErrorCode:=0;

	stStopAlarmsLog.Text := 'nSensorStopAlarm';

	IF iReasonStop.0 THEN stStopAlarmsLog.Text := 'data.Alarms.xMotorError';
	ELSIF iReasonStop.1 THEN stStopAlarmsLog.Text := 'data.Alarms.xComsMotorError';
	ELSIF iReasonStop.2 THEN stStopAlarmsLog.Text := 'data.Alarms.xNotReferenced';
	ELSIF iReasonStop.3 THEN stStopAlarmsLog.Text := 'data.Alarms.xIncoherPhotocellSystem';
	ELSIF iReasonStop.4 THEN stStopAlarmsLog.Text := 'data.Alarms.xAlrInvalidAlignmentPosition';
	ELSIF iReasonStop.5 THEN stStopAlarmsLog.Text := 'data.Alarms.xAlrCriticalPhotocellNotAligned';
	END_IF

	gEventLogLoader(EventData := ADR(stStopAlarmsLog));

END_ACTION

ACTION LogCriticalAlarm:

	stCriticalAlarmsLog.Source := ELOG_TYPE_DETECTION;
	stCriticalAlarmsLog.Severity:= ELOG_SEVERITY_ERROR;
	stCriticalAlarmsLog.Facility:= 0;
	stCriticalAlarmsLog.ErrorCode:=0;

	stCriticalAlarmsLog.Text := 'nSensorCriticalAlarm';

	IF iReasonCritical.0 THEN stCriticalAlarmsLog.Text := 'data.Alarms.xPositionOutOfRange';
//	ELSIF iReasonCritical.1 THEN stCriticalAlarmsLog.Text := '';
//	ELSIF iReasonCritical.2 THEN stCriticalAlarmsLog.Text := '';
//	ELSIF iReasonCritical.3 THEN stCriticalAlarmsLog.Text := '';
//	ELSIF iReasonCritical.4 THEN stCriticalAlarmsLog.Text := '';
//	ELSIF iReasonCritical.5 THEN stCriticalAlarmsLog.Text := '';
	END_IF

	gEventLogLoader(EventData := ADR(stCriticalAlarmsLog));

END_ACTION
```
